KUKA KRL program: MyProgram_117().src

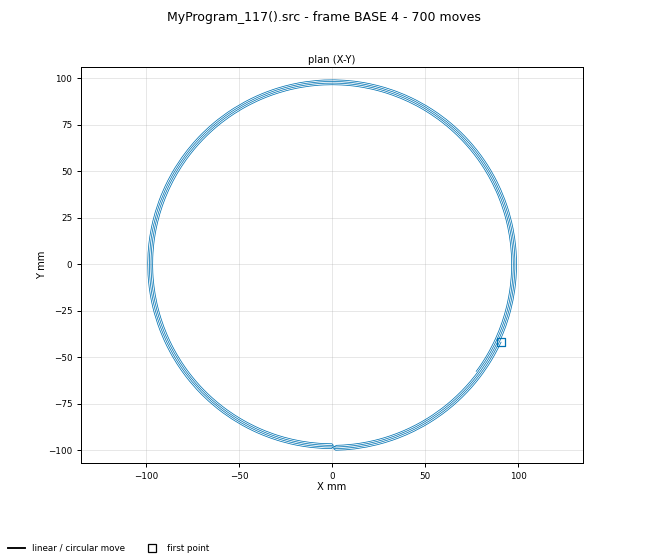
[picture p0: tool path of MyProgram_117().src in frame BASE 4, 700 of 700 moves have a stored position in this frame; points joined in program order, loops and branches not executed]
&ACCESS RVP
&REL 1
&PARAM TEMPLATE = C:\KRC\Roboter\Template\vorgabe
&PARAM EDITMASK = *
DEF MyProgram_117()
; ---- Setting reference (Base) ----
$BASE = BASE_DATA[4]

; --------------------------
; ---- Setting tool (TCP) ----
$TOOL = TOOL_DATA[3]
; --------------------------

$VEL.CP = VEL_APROX_PRINT
Startdeposition()
$VEL.CP = VEL_PRINT
LIN {X 90.8546,Y -41.8961,Z 100,A -29.5079,B 24.9354,C -1.8557,E1 25.1448,E2 114.9492} C_DIS
LIN {X 89.261,Y -45.1921,Z 100,A -32.3169,B 24.9378,C -1.821,E1 25.1412,E2 117.825} C_DIS
LIN {X 87.3886,Y -48.713,Z 100,A -34.4656,B 24.9379,C -1.8197,E1 25.1383,E2 119.9656} C_DIS
LIN {X 85.5953,Y -51.7996,Z 100,A -35.9593,B 24.9368,C -1.8357,E1 25.1362,E2 121.4139} C_DIS
LIN {X 83.9809,Y -54.379,Z 100,A -37.6896,B 24.9371,C -1.8312,E1 25.1336,E2 123.1461} C_DIS
LIN {X 81.1515,Y -58.5183,Z 100,A -40.5595,B 24.9377,C -1.8233,E1 25.129,E2 126.0206} C_DIS
LIN {X 79.2624,Y -61.0507,Z 100,A -42.3506,B 24.938,C -1.8191,E1 25.126,E2 127.813} C_DIS
LIN {X 77.0516,Y -63.8185,Z 100,A -44.3798,B 24.9383,C -1.8138,E1 25.1224,E2 129.8455} C_DIS
LIN {X 74.8748,Y -66.3606,Z 100,A -46.3784,B 24.9389,C -1.8055,E1 25.1187,E2 131.8545} C_DIS
LIN {X 72.5253,Y -68.9207,Z 100,A -48.3686,B 24.9392,C -1.8005,E1 25.1149,E2 133.8478} C_DIS
LIN {X 70.0798,Y -71.4048,Z 100,A -50.3649,B 24.9396,C -1.7957,E1 25.111,E2 135.8471} C_DIS
LIN {X 67.5259,Y -73.824,Z 100,A -52.2794,B 24.9396,C -1.7949,E1 25.1071,E2 137.7558} C_DIS
LIN {X 64.7927,Y -76.2341,Z 100,A -54.4126,B 24.9401,C -1.7883,E1 25.1026,E2 139.8962} C_DIS
LIN {X 61.8717,Y -78.6235,Z 100,A -56.541,B 24.9403,C -1.7848,E1 25.0979,E2 142.0247} C_DIS
LIN {X 59.1319,Y -80.704,Z 100,A -59.2836,B 24.9426,C -1.7507,E1 25.0916,E2 144.8383} C_DIS
LIN {X 55.2065,Y -83.4385,Z 100,A -61.177,B 24.9407,C -1.778,E1 25.0874,E2 146.6607} C_DIS
LIN {X 52.4744,Y -85.1851,Z 100,A -63.1603,B 24.9413,C -1.7695,E1 25.0827,E2 148.6577} C_DIS
LIN {X 49.4197,Y -86.9922,Z 100,A -65.3121,B 24.9419,C -1.7612,E1 25.0774,E2 150.8227} C_DIS
LIN {X 43.9764,Y -89.8668,Z 100,A -68.5455,B 24.9415,C -1.7666,E1 25.0695,E2 154.0344} C_DIS
LIN {X 39.8661,Y -91.7629,Z 100,A -71.8907,B 24.9437,C -1.7338,E1 25.0607,E2 157.4489} C_DIS
LIN {X 35.7477,Y -93.4448,Z 100,A -73.7112,B 24.9421,C -1.758,E1 25.0562,E2 159.2081} C_DIS
LIN {X 32.4545,Y -94.6398,Z 100,A -75.7667,B 24.9424,C -1.7535,E1 25.0507,E2 161.2702} C_DIS
LIN {X 28.1104,Y -96.0182,Z 100,A -78.5161,B 24.9429,C -1.7452,E1 25.0434,E2 164.0343} C_DIS
LIN {X 24.2258,Y -97.0727,Z 100,A -81.6804,B 24.9452,C -1.7105,E1 25.0346,E2 167.276} C_DIS
LIN {X 18.6579,Y -98.2938,Z 100,A -83.3794,B 24.9415,C -1.7666,E1 25.0303,E2 168.84} C_DIS
LIN {X 12.1471,Y -99.3097,Z 100,A -87.4897,B 24.9425,C -1.7511,E1 25.0189,E2 172.9832} C_DIS
LIN {X 7.1479,Y -99.7937,Z 100,A -90.5333,B 24.943,C -1.7433,E1 25.0104,E2 176.0435} C_DIS
LIN {X 1.9327,Y -100.0299,Z 100,A -93.4838,B 24.943,C -1.7437,E1 25.0021,E2 178.9923} C_DIS
LIN {X 1.9327,Y -100.0299,Z 100,A -93.4838,B 24.943,C -1.7437,E1 25.0021,E2 178.9923} C_DIS
Enddeposition()
LIN {X 0.6913,Y -99.1652,Z 100,A -93.9796,B 24.9415,C -1.767,E1 25.0009,E2 179.4329} C_DIS
Startdeposition()
$VEL.CP = VEL_PRINT
LIN {X 6.2659,Y -98.9734,Z 100,A -90.3547,B 24.9404,C -1.7829,E1 25.0111,E2 175.771} C_DIS
LIN {X 9.1996,Y -98.743,Z 100,A -88.1393,B 24.939,C -1.8033,E1 25.0174,E2 173.5087} C_DIS
LIN {X 12.9587,Y -98.3206,Z 100,A -85.2245,B 24.937,C -1.8326,E1 25.0257,E2 170.5267} C_DIS
LIN {X 18.458,Y -97.4382,Z 100,A -83.3272,B 24.9403,C -1.7846,E1 25.0306,E2 168.7453} C_DIS
LIN {X 23.319,Y -96.3902,Z 100,A -80.2469,B 24.9396,C -1.7951,E1 25.039,E2 165.6443} C_DIS
LIN {X 26.3077,Y -95.6187,Z 100,A -78.5649,B 24.9397,C -1.7931,E1 25.0435,E2 163.9697} C_DIS
LIN {X 30.9499,Y -94.2184,Z 100,A -75.585,B 24.9391,C -1.8032,E1 25.0515,E2 160.9713} C_DIS
LIN {X 34.1098,Y -93.1201,Z 100,A -73.9959,B 24.9398,C -1.7925,E1 25.0556,E2 159.4108} C_DIS
LIN {X 40.541,Y -90.5057,Z 100,A -69.6647,B 24.9386,C -1.8105,E1 25.0669,E2 155.0468} C_DIS
LIN {X 43.8774,Y -88.9361,Z 100,A -67.6389,B 24.9386,C -1.8099,E1 25.072,E2 153.0279} C_DIS
LIN {X 46.0291,Y -87.8418,Z 100,A -66.2942,B 24.9386,C -1.8103,E1 25.0753,E2 151.686} C_DIS
LIN {X 49.9401,Y -85.6805,Z 100,A -63.5045,B 24.9377,C -1.823,E1 25.0821,E2 148.8744} C_DIS
LIN {X 52.9459,Y -83.8557,Z 100,A -61.6939,B 24.938,C -1.8182,E1 25.0864,E2 147.0809} C_DIS
LIN {X 57.7115,Y -80.6487,Z 100,A -58.2792,B 24.9373,C -1.8286,E1 25.0943,E2 143.6532} C_DIS
LIN {X 59.9569,Y -78.9951,Z 100,A -56.5708,B 24.9368,C -1.8358,E1 25.0981,E2 141.9339} C_DIS
LIN {X 62.7275,Y -76.8128,Z 100,A -54.5611,B 24.9366,C -1.8392,E1 25.1025,E2 139.9238} C_DIS
LIN {X 65.4078,Y -74.5432,Z 100,A -52.5255,B 24.9363,C -1.8441,E1 25.1068,E2 137.8846} C_DIS
LIN {X 68.1055,Y -72.0868,Z 100,A -50.4771,B 24.9361,C -1.8467,E1 25.111,E2 135.8384} C_DIS
LIN {X 70.6086,Y -69.6365,Z 100,A -48.5177,B 24.9359,C -1.8491,E1 25.1149,E2 133.8817} C_DIS
LIN {X 73.1184,Y -66.9964,Z 100,A -46.4051,B 24.9355,C -1.8547,E1 25.1189,E2 131.7651} C_DIS
LIN {X 75.5655,Y -64.2237,Z 100,A -44.3231,B 24.9353,C -1.858,E1 25.1227,E2 129.6846} C_DIS
LIN {X 77.8109,Y -61.4839,Z 100,A -42.25,B 24.9348,C -1.8645,E1 25.1264,E2 127.6058} C_DIS
LIN {X 79.842,Y -58.8231,Z 100,A -40.4207,B 24.9348,C -1.8656,E1 25.1294,E2 125.7828} C_DIS
LIN {X 81.2965,Y -56.7955,Z 100,A -38.5075,B 24.9331,C -1.8885,E1 25.1326,E2 123.8247} C_DIS
LIN {X 83.0913,Y -54.1382,Z 100,A -36.9749,B 24.9337,C -1.8808,E1 25.1349,E2 122.318} C_DIS
LIN {X 84.6691,Y -51.633,Z 100,A -34.534,B 24.9312,C -1.9153,E1 25.1385,E2 119.8081} C_DIS
LIN {X 87.0569,Y -47.497,Z 100,A -32.9217,B 24.934,C -1.877,E1 25.1406,E2 118.2946} C_DIS
LIN {X 89.1564,Y -43.4308,Z 100,A -29.8964,B 24.9323,C -1.9001,E1 25.1444,E2 115.2308} C_DIS
LIN {X 90.6651,Y -40.1874,Z 100,A -27.4278,B 24.9307,C -1.9227,E1 25.1473,E2 112.7224} C_DIS
LIN {X 92.0383,Y -36.9323,Z 100,A -25.8511,B 24.9316,C -1.9101,E1 25.1489,E2 111.1841} C_DIS
LIN {X 93.3981,Y -33.3451,Z 100,A -23.5352,B 24.9308,C -1.921,E1 25.1511,E2 108.8554} C_DIS
LIN {X 95.0827,Y -28.1796,Z 100,A -20.5952,B 24.9307,C -1.9228,E1 25.1536,E2 105.9278} C_DIS
LIN {X 95.9761,Y -24.9697,Z 100,A -18.685,B 24.9303,C -1.9283,E1 25.155,E2 104.0156} C_DIS
LIN {X 97.2767,Y -19.2966,Z 100,A -15.4761,B 24.93,C -1.9328,E1 25.1569,E2 100.8147} C_DIS
LIN {X 98.201,Y -13.834,Z 100,A -12.0909,B 24.9287,C -1.9505,E1 25.1585,E2 97.4077} C_DIS
LIN {X 98.5903,Y -10.7206,Z 100,A -9.9416,B 24.9272,C -1.97,E1 25.1591,E2 95.2251} C_DIS
LIN {X 98.886,Y -7.5176,Z 100,A -7.8658,B 24.9261,C -1.9849,E1 25.1595,E2 93.1265} C_DIS
LIN {X 99.1121,Y -3.4295,Z 100,A -6.1235,B 24.9274,C -1.9672,E1 25.1597,E2 91.4364} C_DIS
LIN {X 99.1305,Y 2.8285,Z 100,A -1.9325,B 24.9248,C -2.0022,E1 25.1596,E2 87.1877} C_DIS
LIN {X 98.9312,Y 6.8905,Z 100,A -0.1687,B 24.9261,C -1.9859,E1 25.1593,E2 85.4728} C_DIS
LIN {X 98.7353,Y 9.2834,Z 100,A 1.9576,B 24.9235,C -2.0204,E1 25.1587,E2 83.2778} C_DIS
LIN {X 98.1786,Y 13.9922,Z 100,A 3.4043,B 24.9267,C -1.9767,E1 25.1582,E2 81.9425} C_DIS
LIN {X 97.3147,Y 19.0993,Z 100,A 6.8499,B 24.9247,C -2.0042,E1 25.1565,E2 78.4524} C_DIS
LIN {X 96.5792,Y 22.5236,Z 100,A 9.8653,B 24.9211,C -2.0507,E1 25.1546,E2 75.3448} C_DIS
LIN {X 95.1729,Y 27.8757,Z 100,A 12.0003,B 24.9237,C -2.0174,E1 25.153,E2 73.3006} C_DIS
LIN {X 94.2802,Y 30.7591,Z 100,A 13.8408,B 24.923,C -2.0265,E1 25.1514,E2 71.449} C_DIS
LIN {X 92.9322,Y 34.6224,Z 100,A 16.1677,B 24.9226,C -2.032,E1 25.1492,E2 69.1222} C_DIS
LIN {X 90.6792,Y 40.1549,Z 100,A 19.4045,B 24.9225,C -2.0334,E1 25.1458,E2 65.8999} C_DIS
LIN {X 88.6792,Y 44.3956,Z 100,A 22.1934,B 24.9216,C -2.0442,E1 25.1424,E2 63.1005} C_DIS
LIN {X 87.2725,Y 47.0996,Z 100,A 24.1381,B 24.9207,C -2.0563,E1 25.1398,E2 61.1374} C_DIS
LIN {X 85.3146,Y 50.5593,Z 100,A 26.3186,B 24.9206,C -2.0579,E1 25.1368,E2 58.9645} C_DIS
LIN {X 83.6341,Y 53.2941,Z 100,A 28.1593,B 24.9203,C -2.0622,E1 25.134,E2 57.1229} C_DIS
LIN {X 82.0137,Y 55.7549,Z 100,A 30.2378,B 24.9188,C -2.0814,E1 25.1307,E2 55.0092} C_DIS
LIN {X 80.1035,Y 58.466,Z 100,A 31.6874,B 24.9198,C -2.0677,E1 25.1284,E2 53.599} C_DIS
LIN {X 77.9344,Y 61.3277,Z 100,A 33.816,B 24.9193,C -2.0749,E1 25.1248,E2 51.4636} C_DIS
LIN {X 75.5962,Y 64.1876,Z 100,A 35.6617,B 24.9198,C -2.0686,E1 25.1215,E2 49.6412} C_DIS
LIN {X 73.8444,Y 66.1954,Z 100,A 37.9636,B 24.9171,C -2.102,E1 25.1171,E2 47.2706} C_DIS
LIN {X 71.3218,Y 68.906,Z 100,A 39.5535,B 24.9185,C -2.0851,E1 25.1141,E2 45.7275} C_DIS
LIN {X 69.2349,Y 71.0047,Z 100,A 41.4391,B 24.9176,C -2.0956,E1 25.1103,E2 43.8251} C_DIS
LIN {X 66.2722,Y 73.7756,Z 100,A 43.5685,B 24.9179,C -2.092,E1 25.106,E2 41.7128} C_DIS
LIN {X 63.6338,Y 76.0636,Z 100,A 45.9997,B 24.9163,C -2.112,E1 25.1007,E2 39.2438} C_DIS
LIN {X 61.144,Y 78.0795,Z 100,A 48.2904,B 24.9147,C -2.1325,E1 25.0956,E2 36.913} C_DIS
LIN {X 57.2387,Y 80.9861,Z 100,A 50.1264,B 24.9173,C -2.0994,E1 25.0916,E2 35.1617} C_DIS
LIN {X 54.0365,Y 83.1576,Z 100,A 52.6018,B 24.9163,C -2.1123,E1 25.0858,E2 32.6641} C_DIS
LIN {X 50.8122,Y 85.1651,Z 100,A 54.7198,B 24.9163,C -2.1126,E1 25.0808,E2 30.5519} C_DIS
LIN {X 45.3585,Y 88.19,Z 100,A 58.2162,B 24.9163,C -2.1134,E1 25.0722,E2 27.0637} C_DIS
LIN {X 42.553,Y 89.5782,Z 100,A 60.1676,B 24.9156,C -2.1211,E1 25.0673,E2 25.0993} C_DIS
LIN {X 38.7954,Y 91.2679,Z 100,A 62.5974,B 24.9153,C -2.1256,E1 25.061,E2 22.6647} C_DIS
LIN {X 35.0727,Y 92.7616,Z 100,A 64.7142,B 24.9157,C -2.1203,E1 25.0556,E2 20.5651} C_DIS
LIN {X 32.749,Y 93.6073,Z 100,A 66.4711,B 24.9146,C -2.1339,E1 25.0509,E2 18.7794} C_DIS
LIN {X 28.3562,Y 95.0303,Z 100,A 68.8789,B 24.9152,C -2.1262,E1 25.0445,E2 16.3944} C_DIS
LIN {X 24.5316,Y 96.0887,Z 100,A 71.9667,B 24.9127,C -2.1575,E1 25.036,E2 13.2371} C_DIS
LIN {X 19.8131,Y 97.1714,Z 100,A 73.8566,B 24.9153,C -2.1249,E1 25.031,E2 11.427} C_DIS
LIN {X 16.7703,Y 97.7433,Z 100,A 75.4869,B 24.9157,C -2.1197,E1 25.0266,E2 9.8108} C_DIS
LIN {X 12.2429,Y 98.4133,Z 100,A 78.5022,B 24.9146,C -2.134,E1 25.0182,E2 6.7641} C_DIS
LIN {X 7.0795,Y 98.9184,Z 100,A 81.1159,B 24.9157,C -2.1202,E1 25.011,E2 4.1847} C_DIS
LIN {X 1.4329,Y 99.1611,Z 100,A 84.378,B 24.9157,C -2.1198,E1 25.0019,E2 0.9244} C_DIS
LIN {X -4.0931,Y 99.0863,Z 100,A 87.4521,B 24.9161,C -2.1146,E1 24.9934,E2 -2.1376} C_DIS
LIN {X -7.6767,Y 98.8733,Z 100,A 90.1777,B 24.9143,C -2.1373,E1 24.9856,E2 -4.9181} C_DIS
LIN {X -14.3965,Y 98.1211,Z 100,A 93.8164,B 24.9153,C -2.1253,E1 24.9756,E2 -8.5308} C_DIS
LIN {X -17.8618,Y 97.5493,Z 100,A 96.4541,B 24.9137,C -2.1457,E1 24.9682,E2 -11.2196} C_DIS
LIN {X -21.8344,Y 96.7384,Z 100,A 97.9981,B 24.9161,C -2.115,E1 24.9642,E2 -12.6926} C_DIS
LIN {X -25.5325,Y 95.8281,Z 100,A 100.4259,B 24.9156,C -2.1209,E1 24.9576,E2 -15.1379} C_DIS
LIN {X -29.0848,Y 94.8102,Z 100,A 102.2357,B 24.9167,C -2.1071,E1 24.9528,E2 -16.9178} C_DIS
LIN {X -31.6314,Y 93.9908,Z 100,A 104.1295,B 24.9159,C -2.1175,E1 24.9477,E2 -18.84} C_DIS
LIN {X -35.1644,Y 92.7269,Z 100,A 106.1336,B 24.9166,C -2.1089,E1 24.9425,E2 -20.8278} C_DIS
LIN {X -37.7966,Y 91.6861,Z 100,A 107.8796,B 24.9165,C -2.1105,E1 24.9379,E2 -22.5814} C_DIS
LIN {X -40.7171,Y 90.4264,Z 100,A 110.1476,B 24.9155,C -2.123,E1 24.9321,E2 -24.8844} C_DIS
LIN {X -43.672,Y 89.0374,Z 100,A 111.6554,B 24.9168,C -2.1067,E1 24.9284,E2 -26.3574} C_DIS
LIN {X -46.915,Y 87.3726,Z 100,A 113.5154,B 24.9177,C -2.0946,E1 24.9238,E2 -28.1937} C_DIS
LIN {X -53.0828,Y 83.7697,Z 100,A 117.9867,B 24.9174,C -2.0989,E1 24.9131,E2 -32.6891} C_DIS
LIN {X -56.3961,Y 81.574,Z 100,A 120.2522,B 24.9178,C -2.0934,E1 24.9078,E2 -34.9489} C_DIS
LIN {X -61.3368,Y 77.9272,Z 100,A 123.7519,B 24.9185,C -2.0843,E1 24.9,E2 -38.4395} C_DIS
LIN {X -63.4455,Y 76.22,Z 100,A 125.9799,B 24.917,C -2.1036,E1 24.8951,E2 -40.722} C_DIS
LIN {X -66.6139,Y 73.4693,Z 100,A 128.4285,B 24.9174,C -2.0988,E1 24.8901,E2 -43.169} C_DIS
LIN {X -69.5784,Y 70.666,Z 100,A 130.0947,B 24.9197,C -2.0695,E1 24.8869,E2 -44.7722} C_DIS
LIN {X -71.8411,Y 68.3668,Z 100,A 132.6576,B 24.9182,C -2.0888,E1 24.8818,E2 -47.3923} C_DIS
LIN {X -74.5581,Y 65.3907,Z 100,A 134.5074,B 24.9199,C -2.0665,E1 24.8785,E2 -49.1973} C_DIS
LIN {X -77.9352,Y 61.3267,Z 100,A 137.3121,B 24.9212,C -2.0501,E1 24.8736,E2 -51.9759} C_DIS
LIN {X -80.8016,Y 57.4972,Z 100,A 140.3008,B 24.9212,C -2.0502,E1 24.8686,E2 -54.9793} C_DIS
LIN {X -84.438,Y 52.0134,Z 100,A 144.0835,B 24.9221,C -2.0388,E1 24.8629,E2 -58.7539} C_DIS
LIN {X -86.0785,Y 49.2477,Z 100,A 146.7197,B 24.9204,C -2.0599,E1 24.8591,E2 -61.4541} C_DIS
LIN {X -88.337,Y 45.071,Z 100,A 148.636,B 24.9232,C -2.0238,E1 24.8568,E2 -63.2946} C_DIS
LIN {X -89.8728,Y 41.925,Z 100,A 150.3939,B 24.9243,C -2.0089,E1 24.8547,E2 -65.0264} C_DIS
LIN {X -91.9957,Y 37.0345,Z 100,A 154.0806,B 24.9235,C -2.0198,E1 24.8506,E2 -68.7595} C_DIS
LIN {X -93.141,Y 34.0526,Z 100,A 156.8724,B 24.9215,C -2.0462,E1 24.8479,E2 -71.6302} C_DIS
LIN {X -95.0967,Y 28.1325,Z 100,A 158.9789,B 24.9262,C -1.9844,E1 24.8463,E2 -73.6012} C_DIS
LIN {X -96.3633,Y 23.4293,Z 100,A 162.1051,B 24.9261,C -1.9858,E1 24.844,E2 -76.7492} C_DIS
LIN {X -97.147,Y 19.9317,Z 100,A 164.1597,B 24.9266,C -1.9787,E1 24.8428,E2 -78.7988} C_DIS
LIN {X -98.0211,Y 15.0562,Z 100,A 167.0727,B 24.9271,C -1.9712,E1 24.8415,E2 -81.7113} C_DIS
LIN {X -98.5567,Y 11.0293,Z 100,A 170.3255,B 24.9254,C -1.9941,E1 24.8404,E2 -85.0382} C_DIS
LIN {X -98.9855,Y 6.0807,Z 100,A 172.357,B 24.9282,C -1.9566,E1 24.84,E2 -86.9924} C_DIS
LIN {X -99.1342,Y 2.7095,Z 100,A 174.2253,B 24.9289,C -1.9476,E1 24.8398,E2 -88.8505} C_DIS
LIN {X -99.1684,Y 0.6951,Z 100,A 175.7702,B 24.9282,C -1.9566,E1 24.8398,E2 -90.4262} C_DIS
LIN {X -99.0153,Y -5.5482,Z 100,A 179.0512,B 24.9299,C -1.9341,E1 24.8401,E2 -93.6731} C_DIS
LIN {X -98.7637,Y -8.9753,Z 100,A -178.3436,B 24.9288,C -1.9486,E1 24.8408,E2 -96.3287} C_DIS
LIN {X -98.3563,Y -12.6829,Z 100,A -176.6482,B 24.9304,C -1.9263,E1 24.8413,E2 -97.981} C_DIS
LIN {X -97.8334,Y -16.2313,Z 100,A -174.6127,B 24.931,C -1.9185,E1 24.8422,E2 -100.0101} C_DIS
LIN {X -97.2266,Y -19.544,Z 100,A -172.613,B 24.9313,C -1.9143,E1 24.8433,E2 -102.0114} C_DIS
LIN {X -96.4078,Y -23.2471,Z 100,A -170.4736,B 24.9319,C -1.9058,E1 24.8446,E2 -104.1431} C_DIS
LIN {X -95.661,Y -26.151,Z 100,A -168.6012,B 24.9319,C -1.9052,E1 24.846,E2 -106.0251} C_DIS
LIN {X -93.8161,Y -32.1464,Z 100,A -165.0105,B 24.9328,C -1.8932,E1 24.849,E2 -109.6076} C_DIS
LIN {X -92.5501,Y -35.6314,Z 100,A -161.8525,B 24.9308,C -1.9216,E1 24.8523,E2 -112.8513} C_DIS
LIN {X -90.3767,Y -40.8274,Z 100,A -159.6526,B 24.934,C -1.8762,E1 24.8546,E2 -114.955} C_DIS
LIN {X -88.9026,Y -43.9448,Z 100,A -157.6433,B 24.9344,C -1.8712,E1 24.8571,E2 -116.9632} C_DIS
LIN {X -87.2503,Y -47.1404,Z 100,A -155.5837,B 24.9348,C -1.8648,E1 24.8598,E2 -119.0186} C_DIS
LIN {X -85.9838,Y -49.4125,Z 100,A -153.8216,B 24.9345,C -1.8697,E1 24.8622,E2 -120.8013} C_DIS
LIN {X -83.428,Y -53.6152,Z 100,A -150.9996,B 24.935,C -1.8616,E1 24.8664,E2 -123.6184} C_DIS
LIN {X -81.1676,Y -56.9811,Z 100,A -148.8483,B 24.9359,C -1.8491,E1 24.8698,E2 -125.7505} C_DIS
LIN {X -78.917,Y -60.0583,Z 100,A -146.3568,B 24.9356,C -1.8536,E1 24.874,E2 -128.2649} C_DIS
LIN {X -76.6092,Y -62.9772,Z 100,A -143.3514,B 24.9338,C -1.8785,E1 24.8795,E2 -131.3435} C_DIS
LIN {X -72.8133,Y -67.3289,Z 100,A -141.0169,B 24.9368,C -1.8359,E1 24.8837,E2 -133.5869} C_DIS
LIN {X -70.4028,Y -69.8449,Z 100,A -138.0223,B 24.9347,C -1.8662,E1 24.8898,E2 -136.6663} C_DIS
LIN {X -66.3283,Y -73.7253,Z 100,A -135.8013,B 24.9377,C -1.8232,E1 24.8941,E2 -138.7941} C_DIS
LIN {X -61.8773,Y -77.5,Z 100,A -132.2172,B 24.9377,C -1.8243,E1 24.9019,E2 -142.3943} C_DIS
LIN {X -58.6752,Y -79.9503,Z 100,A -129.7231,B 24.9375,C -1.8261,E1 24.9075,E2 -144.9016} C_DIS
LIN {X -53.7609,Y -83.3345,Z 100,A -126.6443,B 24.9388,C -1.8075,E1 24.9145,E2 -147.9462} C_DIS
LIN {X -48.5279,Y -86.4864,Z 100,A -123.0861,B 24.939,C -1.8034,E1 24.9231,E2 -151.5055} C_DIS
LIN {X -45.4862,Y -88.1248,Z 100,A -121.0314,B 24.939,C -1.8029,E1 24.9282,E2 -153.5647} C_DIS
LIN {X -42.6776,Y -89.5183,Z 100,A -119.3698,B 24.9396,C -1.7953,E1 24.9323,E2 -155.2127} C_DIS
LIN {X -40.5018,Y -90.5234,Z 100,A -117.7985,B 24.9392,C -1.8005,E1 24.9363,E2 -156.8001} C_DIS
LIN {X -37.1909,Y -91.9331,Z 100,A -115.8808,B 24.9398,C -1.7925,E1 24.9413,E2 -158.7032} C_DIS
LIN {X -33.2428,Y -93.4333,Z 100,A -113.2446,B 24.9394,C -1.7974,E1 24.9482,E2 -161.3564} C_DIS
LIN {X -29.3727,Y -94.7209,Z 100,A -111.0463,B 24.94,C -1.7899,E1 24.954,E2 -163.5408} C_DIS
LIN {X -27.2455,Y -95.3548,Z 100,A -108.7966,B 24.9376,C -1.8246,E1 24.9603,E2 -165.8764} C_DIS
LIN {X -22.3273,Y -96.6245,Z 100,A -106.7888,B 24.94,C -1.7888,E1 24.9655,E2 -167.8019} C_DIS
LIN {X -19.3944,Y -97.2573,Z 100,A -104.4465,B 24.9386,C -1.8105,E1 24.9721,E2 -170.1985} C_DIS
LIN {X -15.6093,Y -97.9356,Z 100,A -102.0586,B 24.9382,C -1.8161,E1 24.9787,E2 -172.6019} C_DIS
LIN {X -11.1761,Y -98.5395,Z 100,A -100.1508,B 24.9399,C -1.7905,E1 24.9838,E2 -174.4501} C_DIS
LIN {X -4.9792,Y -99.0465,Z 100,A -96.6781,B 24.9402,C -1.786,E1 24.9935,E2 -177.9135} C_DIS
LIN {X -0.5004,Y -99.1694,Z 100,A -94.031,B 24.94,C -1.7886,E1 25.0009,E2 -180.5671} C_DIS
LIN {X -0.5004,Y -99.1694,Z 100,A -94.031,B 24.94,C -1.7886,E1 25.0009,E2 -180.5671} C_DIS
Enddeposition()
LIN {X 0.7031,Y -98.2806,Z 100,A -94.8995,B 24.9428,C -1.7469,E1 24.9982,E2 -179.5997} C_DIS
Startdeposition()
$VEL.CP = VEL_PRINT
LIN {X -3.7844,Y -98.2208,Z 100,A -96.6689,B 24.9408,C -1.777,E1 24.9935,E2 -177.9015} C_DIS
LIN {X -9.0806,Y -97.8724,Z 100,A -99.5035,B 24.9402,C -1.7864,E1 24.9856,E2 -175.088} C_DIS
LIN {X -12.0024,Y -97.5572,Z 100,A -101.792,B 24.9416,C -1.7658,E1 24.9791,E2 -172.7492} C_DIS
LIN {X -15.3506,Y -97.0872,Z 100,A -103.9453,B 24.942,C -1.7597,E1 24.9731,E2 -170.5797} C_DIS
LIN {X -19.3218,Y -96.376,Z 100,A -105.9871,B 24.9412,C -1.7717,E1 24.9676,E2 -168.5641} C_DIS
LIN {X -22.607,Y -95.6589,Z 100,A -108.4713,B 24.9423,C -1.7541,E1 24.9607,E2 -166.0347} C_DIS
LIN {X -25.966,Y -94.8016,Z 100,A -109.8291,B 24.9407,C -1.7788,E1 24.9572,E2 -164.7335} C_DIS
LIN {X -28.3424,Y -94.1187,Z 100,A -111.4726,B 24.9411,C -1.7726,E1 24.9528,E2 -163.0726} C_DIS
LIN {X -31.6213,Y -93.0677,Z 100,A -114.2445,B 24.9428,C -1.7474,E1 24.9453,E2 -160.2357} C_DIS
LIN {X -35.9301,Y -91.4903,Z 100,A -116.1039,B 24.9407,C -1.7784,E1 24.9406,E2 -158.4459} C_DIS
LIN {X -40.2807,Y -89.6601,Z 100,A -118.9222,B 24.9407,C -1.779,E1 24.9334,E2 -155.6224} C_DIS
LIN {X -43.3286,Y -88.2282,Z 100,A -120.8746,B 24.9405,C -1.7816,E1 24.9284,E2 -153.6714} C_DIS
LIN {X -46.1911,Y -86.7642,Z 100,A -122.6869,B 24.9402,C -1.7862,E1 24.924,E2 -151.8649} C_DIS
LIN {X -48.8551,Y -85.2916,Z 100,A -124.7909,B 24.9408,C -1.7773,E1 24.9188,E2 -149.7336} C_DIS
LIN {X -52.593,Y -83.0409,Z 100,A -127.2914,B 24.9404,C -1.7825,E1 24.9129,E2 -147.2378} C_DIS
LIN {X -56.3842,Y -80.5133,Z 100,A -129.9455,B 24.9401,C -1.787,E1 24.9068,E2 -144.5853} C_DIS
LIN {X -59.6748,Y -78.106,Z 100,A -133.5265,B 24.9426,C -1.7506,E1 24.8986,E2 -140.9047} C_DIS
LIN {X -64.9815,Y -73.7499,Z 100,A -135.4992,B 24.9374,C -1.8268,E1 24.8948,E2 -139.1058} C_DIS
LIN {X -70.1765,Y -68.8247,Z 100,A -140.036,B 24.9377,C -1.8228,E1 24.8855,E2 -134.5407} C_DIS
LIN {X -75.4021,Y -63.0561,Z 100,A -144.6109,B 24.9371,C -1.8317,E1 24.877,E2 -129.9666} C_DIS
LIN {X -79.3284,Y -58.0385,Z 100,A -148.5605,B 24.9371,C -1.8327,E1 24.8702,E2 -126.0007} C_DIS
LIN {X -81.2404,Y -55.331,Z 100,A -150.6432,B 24.9371,C -1.8325,E1 24.8668,E2 -123.9073} C_DIS
LIN {X -82.7159,Y -53.0993,Z 100,A -152.646,B 24.9378,C -1.8219,E1 24.8638,E2 -121.8691} C_DIS
LIN {X -84.5723,Y -50.0898,Z 100,A -154.1854,B 24.9362,C -1.8446,E1 24.8616,E2 -120.3758} C_DIS
LIN {X -85.8025,Y -47.952,Z 100,A -155.6566,B 24.936,C -1.8473,E1 24.8596,E2 -118.9035} C_DIS
LIN {X -87.4778,Y -44.8231,Z 100,A -157.7262,B 24.9356,C -1.853,E1 24.8569,E2 -116.8363} C_DIS
LIN {X -89.0012,Y -41.717,Z 100,A -159.7411,B 24.9352,C -1.8587,E1 24.8545,E2 -114.8241} C_DIS
LIN {X -91.1623,Y -36.7559,Z 100,A -162.6115,B 24.9339,C -1.8771,E1 24.8514,E2 -111.9818} C_DIS
LIN {X -92.5847,Y -33.0118,Z 100,A -165.735,B 24.9353,C -1.8581,E1 24.8483,E2 -108.7953} C_DIS
LIN {X -93.6148,Y -29.9623,Z 100,A -167.1224,B 24.9338,C -1.8796,E1 24.8471,E2 -107.4514} C_DIS
LIN {X -94.3373,Y -27.6054,Z 100,A -168.7403,B 24.9338,C -1.8781,E1 24.8458,E2 -105.8204} C_DIS
LIN {X -95.2127,Y -24.4133,Z 100,A -170.5413,B 24.9332,C -1.8882,E1 24.8445,E2 -104.033} C_DIS
LIN {X -96.017,Y -21.0287,Z 100,A -172.6216,B 24.9328,C -1.8927,E1 24.8432,E2 -101.9513} C_DIS
LIN {X -96.7295,Y -17.4606,Z 100,A -174.7143,B 24.9323,C -1.9002,E1 24.8421,E2 -99.8642} C_DIS
LIN {X -97.214,Y -14.5307,Z 100,A -176.6315,B 24.9323,C -1.8996,E1 24.8413,E2 -97.9341} C_DIS
LIN {X -97.7927,Y -9.9071,Z 100,A -179.13,B 24.9312,C -1.9153,E1 24.8405,E2 -95.4581} C_DIS
LIN {X -98.0751,Y -6.5381,Z 100,A 178.7822,B 24.931,C -1.9178,E1 24.8401,E2 -93.3636} C_DIS
LIN {X -98.2689,Y -2.1956,Z 100,A 176.167,B 24.9307,C -1.9233,E1 24.8398,E2 -90.7458} C_DIS
LIN {X -98.2774,Y 1.7359,Z 100,A 173.9513,B 24.9299,C -1.9331,E1 24.8398,E2 -88.5403} C_DIS
LIN {X -98.1668,Y 4.9918,Z 100,A 171.8896,B 24.9299,C -1.9339,E1 24.8401,E2 -86.468} C_DIS
LIN {X -97.7338,Y 10.4695,Z 100,A 168.7137,B 24.9291,C -1.9451,E1 24.8409,E2 -83.2999} C_DIS
LIN {X -97.2936,Y 13.9796,Z 100,A 166.2454,B 24.9295,C -1.9387,E1 24.8418,E2 -80.8014} C_DIS
LIN {X -96.7553,Y 17.3167,Z 100,A 164.5822,B 24.9284,C -1.9549,E1 24.8426,E2 -79.167} C_DIS
LIN {X -96.0221,Y 21.0051,Z 100,A 162.5374,B 24.9275,C -1.9666,E1 24.8438,E2 -77.1382} C_DIS
LIN {X -94.3008,Y 27.7287,Z 100,A 157.9594,B 24.9278,C -1.9622,E1 24.8471,E2 -72.523} C_DIS
LIN {X -93.2688,Y 31.023,Z 100,A 156.3612,B 24.9264,C -1.9819,E1 24.8485,E2 -70.9626} C_DIS
LIN {X -92.3152,Y 33.7546,Z 100,A 154.6854,B 24.9259,C -1.9874,E1 24.8501,E2 -69.2905} C_DIS
LIN {X -89.5641,Y 40.4937,Z 100,A 150.7004,B 24.9243,C -2.0087,E1 24.8543,E2 -65.3343} C_DIS
LIN {X -88.5287,Y 42.7101,Z 100,A 149.0427,B 24.9246,C -2.0054,E1 24.8563,E2 -63.6597} C_DIS
LIN {X -86.1069,Y 47.4057,Z 100,A 146.0899,B 24.9236,C -2.0186,E1 24.8601,E2 -60.7225} C_DIS
LIN {X -84.5142,Y 50.1881,Z 100,A 143.9706,B 24.9238,C -2.0158,E1 24.8631,E2 -58.5855} C_DIS
LIN {X -81.842,Y 54.438,Z 100,A 140.8042,B 24.9238,C -2.0162,E1 24.8679,E2 -55.4042} C_DIS
LIN {X -78.4434,Y 59.2297,Z 100,A 137.8768,B 24.9218,C -2.0418,E1 24.8726,E2 -52.5236} C_DIS
LIN {X -76.4122,Y 61.8275,Z 100,A 135.6842,B 24.9221,C -2.038,E1 24.8765,E2 -50.3115} C_DIS
LIN {X -74.175,Y 64.4948,Z 100,A 132.7502,B 24.924,C -2.0136,E1 24.882,E2 -47.3061} C_DIS
LIN {X -70.7666,Y 68.2169,Z 100,A 130.8743,B 24.9207,C -2.0559,E1 24.8854,E2 -45.5228} C_DIS
LIN {X -67.8558,Y 71.1124,Z 100,A 128.1822,B 24.9211,C -2.0517,E1 24.8908,E2 -42.8094} C_DIS
LIN {X -64.4484,Y 74.2155,Z 100,A 125.3056,B 24.9211,C -2.0515,E1 24.8968,E2 -39.921} C_DIS
LIN {X -60.7855,Y 77.2437,Z 100,A 122.4919,B 24.9207,C -2.0561,E1 24.9029,E2 -37.1076} C_DIS
LIN {X -57.327,Y 79.8446,Z 100,A 120.5242,B 24.9189,C -2.0798,E1 24.9073,E2 -35.1896} C_DIS
LIN {X -55.6186,Y 81.0455,Z 100,A 119.052,B 24.9194,C -2.0737,E1 24.9107,E2 -33.6977} C_DIS
LIN {X -52.9883,Y 82.7871,Z 100,A 117.2874,B 24.9189,C -2.0797,E1 24.9148,E2 -31.9417} C_DIS
LIN {X -47.8568,Y 85.8556,Z 100,A 113.838,B 24.9183,C -2.0872,E1 24.9231,E2 -28.4997} C_DIS
LIN {X -45.2856,Y 87.2411,Z 100,A 111.7097,B 24.9192,C -2.0756,E1 24.9284,E2 -26.3379} C_DIS
LIN {X -40.5076,Y 89.5578,Z 100,A 109.2375,B 24.9172,C -2.1017,E1 24.9345,E2 -23.9214} C_DIS
LIN {X -37.5307,Y 90.8469,Z 100,A 106.9552,B 24.918,C -2.091,E1 24.9405,E2 -21.6084} C_DIS
LIN {X -34.28,Y 92.123,Z 100,A 104.6053,B 24.9186,C -2.0829,E1 24.9466,E2 -19.2344} C_DIS
LIN {X -30.2573,Y 93.5198,Z 100,A 102.7517,B 24.9167,C -2.1075,E1 24.9514,E2 -17.4359} C_DIS
LIN {X -27.899,Y 94.2502,Z 100,A 101.0737,B 24.9172,C -2.1009,E1 24.9559,E2 -15.7392} C_DIS
LIN {X -24.9823,Y 95.0664,Z 100,A 99.0955,B 24.9177,C -2.0953,E1 24.9613,E2 -13.7448} C_DIS
LIN {X -22.0446,Y 95.7888,Z 100,A 97.2058,B 24.9179,C -2.0926,E1 24.9665,E2 -11.8461} C_DIS
LIN {X -17.9671,Y 96.6384,Z 100,A 94.9122,B 24.9174,C -2.0992,E1 24.9727,E2 -9.5656} C_DIS
LIN {X -14.1589,Y 97.2682,Z 100,A 92.4639,B 24.9178,C -2.0939,E1 24.9795,E2 -7.1025} C_DIS
LIN {X -7.0121,Y 98.043,Z 100,A 88.6789,B 24.9165,C -2.1102,E1 24.99,E2 -3.3542} C_DIS
LIN {X -4.124,Y 98.2062,Z 100,A 86.2458,B 24.9185,C -2.0845,E1 24.9969,E2 -0.8597} C_DIS
LIN {X 0.1184,Y 98.2938,Z 100,A 84.6375,B 24.9161,C -2.1155,E1 25.0012,E2 0.675} C_DIS
LIN {X 5.3634,Y 98.1463,Z 100,A 81.6636,B 24.9158,C -2.1188,E1 25.0095,E2 3.6404} C_DIS
LIN {X 10.6573,Y 97.7142,Z 100,A 78.3393,B 24.9165,C -2.1103,E1 25.0188,E2 6.983} C_DIS
LIN {X 14.5406,Y 97.2121,Z 100,A 75.9614,B 24.9168,C -2.1064,E1 25.0254,E2 9.3684} C_DIS
LIN {X 18.1007,Y 96.613,Z 100,A 73.7692,B 24.9171,C -2.1024,E1 25.0314,E2 11.5675} C_DIS
LIN {X 23.3318,Y 95.4834,Z 100,A 70.8393,B 24.9167,C -2.1077,E1 25.0393,E2 14.481} C_DIS
LIN {X 26.7547,Y 94.5814,Z 100,A 68.7627,B 24.9168,C -2.1058,E1 25.0449,E2 16.5586} C_DIS
LIN {X 32.5393,Y 92.7505,Z 100,A 65.293,B 24.9168,C -2.1054,E1 25.0542,E2 20.0227} C_DIS
LIN {X 35.4757,Y 91.6686,Z 100,A 63.249,B 24.9176,C -2.0956,E1 25.0595,E2 22.0856} C_DIS
LIN {X 38.5242,Y 90.4295,Z 100,A 61.5725,B 24.9171,C -2.1025,E1 25.0638,E2 23.7419} C_DIS
LIN {X 41.7358,Y 88.9925,Z 100,A 59.5129,B 24.9173,C -2.0998,E1 25.069,E2 25.8027} C_DIS
LIN {X 44.4942,Y 87.6458,Z 100,A 57.715,B 24.9175,C -2.0972,E1 25.0735,E2 27.6019} C_DIS
LIN {X 48.3497,Y 85.5804,Z 100,A 55.2562,B 24.9175,C -2.0972,E1 25.0796,E2 30.0539} C_DIS
LIN {X 50.5089,Y 84.3246,Z 100,A 53.2525,B 24.9193,C -2.0746,E1 25.0845,E2 32.1046} C_DIS
LIN {X 55.3469,Y 81.2296,Z 100,A 50.2955,B 24.9186,C -2.0838,E1 25.0913,E2 35.03} C_DIS
LIN {X 61.5543,Y 76.6319,Z 100,A 45.6992,B 24.9195,C -2.0723,E1 25.1016,E2 39.6369} C_DIS
LIN {X 65.1812,Y 73.5739,Z 100,A 43.0592,B 24.9195,C -2.0716,E1 25.1071,E2 42.2682} C_DIS
LIN {X 67.4662,Y 71.4829,Z 100,A 41.3382,B 24.9195,C -2.0712,E1 25.1106,E2 43.9834} C_DIS
LIN {X 69.1978,Y 69.808,Z 100,A 39.8013,B 24.9202,C -2.0632,E1 25.1137,E2 45.5327} C_DIS
LIN {X 73.7304,Y 65.0039,Z 100,A 36.2402,B 24.92,C -2.0656,E1 25.1205,E2 49.0723} C_DIS
LIN {X 75.1292,Y 63.382,Z 100,A 34.6532,B 24.9212,C -2.0498,E1 25.1234,E2 50.6896} C_DIS
LIN {X 77.4684,Y 60.5015,Z 100,A 32.5906,B 24.9213,C -2.0484,E1 25.127,E2 52.7457} C_DIS
LIN {X 79.4717,Y 57.8427,Z 100,A 30.1291,B 24.9232,C -2.0237,E1 25.1311,E2 55.2537} C_DIS
LIN {X 81.7242,Y 54.6165,Z 100,A 27.9606,B 24.9232,C -2.0226,E1 25.1345,E2 57.4142} C_DIS
LIN {X 83.551,Y 51.7766,Z 100,A 26.6735,B 24.9217,C -2.0437,E1 25.1363,E2 58.645} C_DIS
LIN {X 84.9275,Y 49.4888,Z 100,A 24.768,B 24.923,C -2.026,E1 25.139,E2 60.5824} C_DIS
LIN {X 86.6968,Y 46.3184,Z 100,A 22.8747,B 24.9228,C -2.0289,E1 25.1415,E2 62.459} C_DIS
LIN {X 88.02,Y 43.7486,Z 100,A 20.8751,B 24.9241,C -2.012,E1 25.1441,E2 64.4878} C_DIS
LIN {X 90.8782,Y 37.4539,Z 100,A 17.1179,B 24.9241,C -2.011,E1 25.1483,E2 68.2267} C_DIS
LIN {X 92.1336,Y 34.2506,Z 100,A 15.0035,B 24.9249,C -2.0009,E1 25.1504,E2 70.3533} C_DIS
LIN {X 93.5372,Y 30.2034,Z 100,A 12.7575,B 24.9248,C -2.0033,E1 25.1524,E2 72.5811} C_DIS
LIN {X 94.419,Y 27.3279,Z 100,A 10.3232,B 24.9271,C -1.9714,E1 25.1544,E2 75.0767} C_DIS
LIN {X 95.4247,Y 23.5724,Z 100,A 8.6089,B 24.9261,C -1.9859,E1 25.1555,E2 76.7467} C_DIS
LIN {X 96.1788,Y 20.2823,Z 100,A 6.6164,B 24.9266,C -1.9788,E1 25.1567,E2 78.7444} C_DIS
LIN {X 97.1257,Y 15.102,Z 100,A 3.7878,B 24.9266,C -1.9787,E1 25.158,E2 81.5568} C_DIS
LIN {X 97.8014,Y 9.8148,Z 100,A 0.7369,B 24.9272,C -1.971,E1 25.1591,E2 84.6077} C_DIS
LIN {X 97.9699,Y 7.9609,Z 100,A -1.3934,B 24.9304,C -1.9267,E1 25.1596,E2 86.8299} C_DIS
LIN {X 98.2498,Y 2.9056,Z 100,A -3.8008,B 24.9296,C -1.9384,E1 25.1598,E2 89.1955} C_DIS
LIN {X 98.2666,Y -2.3222,Z 100,A -7.1594,B 24.9312,C -1.9164,E1 25.1596,E2 92.5859} C_DIS
LIN {X 98.0706,Y -6.604,Z 100,A -9.0668,B 24.9301,C -1.9314,E1 25.1593,E2 94.4465} C_DIS
LIN {X 97.7923,Y -9.9113,Z 100,A -10.8803,B 24.9301,C -1.9299,E1 25.1588,E2 96.2528} C_DIS
LIN {X 97.3762,Y -13.3986,Z 100,A -12.8572,B 24.9304,C -1.9261,E1 25.1581,E2 98.2271} C_DIS
LIN {X 96.5952,Y -18.1927,Z 100,A -15.6189,B 24.9309,C -1.9198,E1 25.1568,E2 100.9875} C_DIS
LIN {X 95.8023,Y -21.9863,Z 100,A -17.5664,B 24.9305,C -1.9249,E1 25.1557,E2 102.9117} C_DIS
LIN {X 95.2668,Y -24.2028,Z 100,A -19.2956,B 24.932,C -1.9048,E1 25.1545,E2 104.6782} C_DIS
LIN {X 94.3401,Y -27.5962,Z 100,A -21.3698,B 24.9325,C -1.8974,E1 25.1529,E2 106.758} C_DIS
LIN {X 92.5772,Y -33.0331,Z 100,A -24.5314,B 24.9328,C -1.8937,E1 25.1502,E2 109.9105} C_DIS
LIN {X 91.4703,Y -35.981,Z 100,A -26.6773,B 24.934,C -1.8758,E1 25.148,E2 112.0866} C_DIS
LIN {X 90.2134,Y -39.0266,Z 100,A -28.4011,B 24.934,C -1.8777,E1 25.1461,E2 113.7966} C_DIS
LIN {X 88.8249,Y -42.0936,Z 100,A -30.2689,B 24.934,C -1.8754,E1 25.1439,E2 115.6596} C_DIS
LIN {X 86.7798,Y -46.1615,Z 100,A -33.4791,B 24.9361,C -1.8459,E1 25.1397,E2 118.9226} C_DIS
LIN {X 84.9535,Y -49.4416,Z 100,A -35.2648,B 24.9355,C -1.8552,E1 25.1373,E2 120.6771} C_DIS
LIN {X 83.2532,Y -52.2533,Z 100,A -37.067,B 24.9355,C -1.8541,E1 25.1346,E2 122.4726} C_DIS
LIN {X 80.0392,Y -57.0543,Z 100,A -40.3207,B 24.9359,C -1.8492,E1 25.1295,E2 125.7219} C_DIS
LIN {X 77.9042,Y -59.9367,Z 100,A -42.4064,B 24.9363,C -1.8437,E1 25.126,E2 127.8105} C_DIS
LIN {X 75.6641,Y -62.7409,Z 100,A -44.4796,B 24.9366,C -1.8389,E1 25.1224,E2 129.8855} C_DIS
LIN {X 73.3244,Y -65.46,Z 100,A -46.5728,B 24.937,C -1.8335,E1 25.1185,E2 131.9821} C_DIS
LIN {X 70.9022,Y -68.0762,Z 100,A -48.6453,B 24.9373,C -1.8285,E1 25.1145,E2 134.0573} C_DIS
LIN {X 68.498,Y -70.4957,Z 100,A -50.6014,B 24.9376,C -1.8249,E1 25.1107,E2 136.0137} C_DIS
LIN {X 66.1818,Y -72.6743,Z 100,A -52.5606,B 24.9382,C -1.8164,E1 25.1066,E2 137.9849} C_DIS
LIN {X 63.4691,Y -75.055,Z 100,A -54.6194,B 24.9384,C -1.8134,E1 25.1023,E2 140.0429} C_DIS
LIN {X 60.8764,Y -77.1721,Z 100,A -56.5592,B 24.9386,C -1.8095,E1 25.098,E2 141.9844} C_DIS
LIN {X 57.1613,Y -79.9628,Z 100,A -59.5672,B 24.9398,C -1.7924,E1 25.0912,E2 145.0222} C_DIS
LIN {X 52.521,Y -83.0859,Z 100,A -62.286,B 24.9388,C -1.8067,E1 25.0849,E2 147.6983} C_DIS
LIN {X 48.2847,Y -85.6166,Z 100,A -65.0878,B 24.939,C -1.8043,E1 25.0782,E2 150.4972} C_DIS
LIN {X 46.4889,Y -86.605,Z 100,A -66.3783,B 24.9394,C -1.7985,E1 25.075,E2 151.7976} C_DIS
LIN {X 43.821,Y -87.9841,Z 100,A -68.2887,B 24.94,C -1.7896,E1 25.0702,E2 153.724} C_DIS
LIN {X 40.3589,Y -89.6249,Z 100,A -70.4444,B 24.94,C -1.789,E1 25.0648,E2 155.8755} C_DIS
LIN {X 34.7782,Y -91.9344,Z 100,A -73.9799,B 24.9404,C -1.7834,E1 25.0556,E2 159.4161} C_DIS
LIN {X 31.389,Y -93.1461,Z 100,A -76.4454,B 24.9415,C -1.767,E1 25.049,E2 161.9156} C_DIS
LIN {X 27.2718,Y -94.4349,Z 100,A -78.5446,B 24.9406,C -1.7796,E1 25.0435,E2 163.9813} C_DIS
LIN {X 24.0054,Y -95.3175,Z 100,A -80.4943,B 24.9407,C -1.7784,E1 25.0382,E2 165.9308} C_DIS
LIN {X 19.6731,Y -96.3039,Z 100,A -82.9702,B 24.9406,C -1.7803,E1 25.0315,E2 168.399} C_DIS
LIN {X 14.8442,Y -97.1655,Z 100,A -85.9126,B 24.941,C -1.7749,E1 25.0234,E2 171.3509} C_DIS
LIN {X 11.5338,Y -97.6137,Z 100,A -88.5867,B 24.9428,C -1.7471,E1 25.0158,E2 174.0889} C_DIS
LIN {X 7.4408,Y -98.0114,Z 100,A -90.1878,B 24.941,C -1.775,E1 25.0115,E2 175.6232} C_DIS
LIN {X 3.0675,Y -98.2448,Z 100,A -92.8882,B 24.9414,C -1.7686,E1 25.004,E2 178.3378} C_DIS
LIN {X 0.7031,Y -98.2806,Z 100,A -94.8963,B 24.9429,C -1.7456,E1 24.9982,E2 180.4003} C_DIS
Enddeposition()
LIN {X 0.7031,Y -98.2806,Z 100,A -94.8963,B 24.9429,C -1.7456,E1 24.9982,E2 180.4003} C_DIS
Startdeposition()
$VEL.CP = VEL_PRINT
LIN {X 2.3662,Y -97.3877,Z 100,A -92.3362,B 24.938,C -1.8186,E1 25.0059,E2 177.6673} C_DIS
LIN {X 6.0828,Y -97.2259,Z 100,A -89.867,B 24.9372,C -1.8299,E1 25.0128,E2 175.1722} C_DIS
LIN {X 11.2953,Y -96.7577,Z 100,A -87.2335,B 24.9382,C -1.8151,E1 25.02,E2 172.5755} C_DIS
LIN {X 14.5931,Y -96.316,Z 100,A -85.1174,B 24.9377,C -1.8224,E1 25.0259,E2 170.444} C_DIS
LIN {X 18.8716,Y -95.5705,Z 100,A -82.666,B 24.9379,C -1.8206,E1 25.0326,E2 167.9997} C_DIS
LIN {X 22.4997,Y -94.7826,Z 100,A -80.5398,B 24.9379,C -1.8205,E1 25.0384,E2 165.8766} C_DIS
LIN {X 25.5063,Y -94.0164,Z 100,A -78.6278,B 24.9375,C -1.8257,E1 25.0436,E2 163.9553} C_DIS
LIN {X 28.2537,Y -93.2293,Z 100,A -76.9162,B 24.9373,C -1.8287,E1 25.0482,E2 162.2395} C_DIS
LIN {X 31.3954,Y -92.2174,Z 100,A -74.9784,B 24.9372,C -1.831,E1 25.0533,E2 160.3} C_DIS
LIN {X 34.8153,Y -90.9816,Z 100,A -72.7203,B 24.9366,C -1.8384,E1 25.0592,E2 158.0291} C_DIS
LIN {X 38.3497,Y -89.5503,Z 100,A -70.5846,B 24.9367,C -1.8376,E1 25.0647,E2 155.9004} C_DIS
LIN {X 41.6719,Y -88.0535,Z 100,A -68.4217,B 24.9364,C -1.8417,E1 25.0702,E2 153.7334} C_DIS
LIN {X 45.0198,Y -86.3889,Z 100,A -66.3107,B 24.9364,C -1.842,E1 25.0754,E2 151.6274} C_DIS
LIN {X 47.9999,Y -84.7702,Z 100,A -64.4914,B 24.9366,C -1.8388,E1 25.0799,E2 149.821} C_DIS
LIN {X 51.1517,Y -82.9062,Z 100,A -61.7396,B 24.9347,C -1.8659,E1 25.0866,E2 147.0137} C_DIS
LIN {X 53.9186,Y -81.1313,Z 100,A -60.124,B 24.9353,C -1.8574,E1 25.0903,E2 145.4235} C_DIS
LIN {X 59.1251,Y -77.4212,Z 100,A -56.4725,B 24.9351,C -1.861,E1 25.0985,E2 141.7765} C_DIS
LIN {X 62.0144,Y -75.1263,Z 100,A -54.4198,B 24.9351,C -1.8612,E1 25.1029,E2 139.7311} C_DIS
LIN {X 64.6107,Y -72.9063,Z 100,A -52.365,B 24.9346,C -1.8676,E1 25.1073,E2 137.6692} C_DIS
LIN {X 67.2131,Y -70.5147,Z 100,A -50.2348,B 24.9341,C -1.8745,E1 25.1116,E2 135.5315} C_DIS
LIN {X 69.7924,Y -67.9625,Z 100,A -48.1634,B 24.9339,C -1.8773,E1 25.1157,E2 133.4624} C_DIS
LIN {X 72.236,Y -65.3595,Z 100,A -46.0654,B 24.9336,C -1.8825,E1 25.1197,E2 131.3612} C_DIS
LIN {X 74.5705,Y -62.6832,Z 100,A -43.9365,B 24.9331,C -1.8895,E1 25.1235,E2 129.2255} C_DIS
LIN {X 76.8989,Y -59.803,Z 100,A -41.8903,B 24.9331,C -1.8901,E1 25.1271,E2 127.1874} C_DIS
LIN {X 78.4462,Y -57.7572,Z 100,A -40.5699,B 24.9333,C -1.8868,E1 25.1293,E2 125.881} C_DIS
LIN {X 82.435,Y -51.906,Z 100,A -36.1773,B 24.9318,C -1.9074,E1 25.1361,E2 121.4617} C_DIS
LIN {X 85.0688,Y -47.4652,Z 100,A -32.8508,B 24.9303,C -1.9276,E1 25.1408,E2 118.1046} C_DIS
LIN {X 87.2077,Y -43.4107,Z 100,A -30.7121,B 24.9314,C -1.9136,E1 25.1435,E2 116.0103} C_DIS
LIN {X 88.8196,Y -40.0089,Z 100,A -28.3096,B 24.9303,C -1.9277,E1 25.1463,E2 113.5876} C_DIS
LIN {X 90.2695,Y -36.6206,Z 100,A -26.0905,B 24.9297,C -1.9364,E1 25.1487,E2 111.3602} C_DIS
LIN {X 91.4366,Y -33.6012,Z 100,A -24.529,B 24.9303,C -1.9287,E1 25.1502,E2 109.8254} C_DIS
LIN {X 92.414,Y -30.8124,Z 100,A -22.5908,B 24.9293,C -1.942,E1 25.152,E2 107.8668} C_DIS
LIN {X 93.2129,Y -28.3077,Z 100,A -20.8543,B 24.9284,C -1.9544,E1 25.1535,E2 106.1109} C_DIS
LIN {X 94.226,Y -24.7254,Z 100,A -19.0253,B 24.9289,C -1.9471,E1 25.1548,E2 104.3098} C_DIS
LIN {X 94.9148,Y -21.9278,Z 100,A -17.3672,B 24.9286,C -1.951,E1 25.1559,E2 102.6518} C_DIS
LIN {X 95.5534,Y -18.96,Z 100,A -15.537,B 24.9281,C -1.9585,E1 25.1569,E2 100.8147} C_DIS
LIN {X 96.1089,Y -15.898,Z 100,A -13.6888,B 24.9276,C -1.9651,E1 25.1578,E2 98.9618} C_DIS
LIN {X 96.5659,Y -12.8361,Z 100,A -12.0351,B 24.9276,C -1.9643,E1 25.1585,E2 97.3196} C_DIS
LIN {X 96.8812,Y -10.1822,Z 100,A -10.2292,B 24.9266,C -1.9787,E1 25.159,E2 95.4906} C_DIS
LIN {X 97.1753,Y -6.8319,Z 100,A -8.3772,B 24.9265,C -1.9801,E1 25.1595,E2 93.6463} C_DIS
LIN {X 97.3564,Y -3.3981,Z 100,A -6.1921,B 24.9255,C -1.993,E1 25.1597,E2 91.4436} C_DIS
LIN {X 97.4155,Y 0.1709,Z 100,A -4.1085,B 24.9251,C -1.9992,E1 25.1597,E2 89.3579} C_DIS
LIN {X 97.322,Y 4.2516,Z 100,A -1.3909,B 24.9235,C -2.0195,E1 25.1595,E2 86.6086} C_DIS
LIN {X 96.9865,Y 9.1267,Z 100,A 0.877,B 24.9247,C -2.0046,E1 25.159,E2 84.3891} C_DIS
LIN {X 96.4845,Y 13.4331,Z 100,A 3.6212,B 24.9235,C -2.0203,E1 25.1581,E2 81.6241} C_DIS
LIN {X 96.126,Y 15.796,Z 100,A 5.0646,B 24.923,C -2.0263,E1 25.1574,E2 80.1752} C_DIS
LIN {X 95.4897,Y 19.2732,Z 100,A 6.8319,B 24.9235,C -2.0205,E1 25.1565,E2 78.432} C_DIS
LIN {X 94.9117,Y 21.9411,Z 100,A 8.7007,B 24.9223,C -2.0358,E1 25.1554,E2 76.5378} C_DIS
LIN {X 94.2475,Y 24.6418,Z 100,A 10.4761,B 24.9215,C -2.0463,E1 25.1541,E2 74.7478} C_DIS
LIN {X 93.1227,Y 28.5986,Z 100,A 12.6441,B 24.9217,C -2.0437,E1 25.1524,E2 72.5982} C_DIS
LIN {X 92.2301,Y 31.3578,Z 100,A 14.2699,B 24.9215,C -2.0457,E1 25.151,E2 70.977} C_DIS
LIN {X 90.8927,Y 35.0499,Z 100,A 16.793,B 24.9204,C -2.0609,E1 25.1485,E2 68.4322} C_DIS
LIN {X 87.9849,Y 41.8144,Z 100,A 20.966,B 24.9199,C -2.067,E1 25.1438,E2 64.2674} C_DIS
LIN {X 86.4932,Y 44.8204,Z 100,A 23.058,B 24.9191,C -2.0771,E1 25.1412,E2 62.1627} C_DIS
LIN {X 84.7167,Y 48.0935,Z 100,A 25.2194,B 24.9187,C -2.0819,E1 25.1382,E2 60.0012} C_DIS
LIN {X 82.8832,Y 51.1885,Z 100,A 27.4013,B 24.9181,C -2.0901,E1 25.1351,E2 57.8112} C_DIS
LIN {X 80.6689,Y 54.6093,Z 100,A 29.5206,B 24.9184,C -2.0855,E1 25.1318,E2 55.7133} C_DIS
LIN {X 78.84,Y 57.2195,Z 100,A 31.3077,B 24.9184,C -2.0868,E1 25.1289,E2 53.9317} C_DIS
LIN {X 77.0535,Y 59.6022,Z 100,A 33.1679,B 24.9177,C -2.0953,E1 25.1258,E2 52.0604} C_DIS
LIN {X 75.1835,Y 61.9455,Z 100,A 35.1077,B 24.9168,C -2.1063,E1 25.1223,E2 50.1037} C_DIS
LIN {X 69.6309,Y 68.1278,Z 100,A 39.9065,B 24.9162,C -2.1137,E1 25.1133,E2 45.3085} C_DIS
LIN {X 67.2075,Y 70.5202,Z 100,A 41.9739,B 24.9157,C -2.1203,E1 25.1091,E2 43.234} C_DIS
LIN {X 64.321,Y 73.1611,Z 100,A 44.3892,B 24.915,C -2.1293,E1 25.1041,E2 40.8071} C_DIS
LIN {X 61.9707,Y 75.1626,Z 100,A 46.4773,B 24.9139,C -2.1431,E1 25.0995,E2 38.6943} C_DIS
LIN {X 59.1474,Y 77.404,Z 100,A 48.6036,B 24.9135,C -2.1472,E1 25.0948,E2 36.5662} C_DIS
LIN {X 56.1859,Y 79.5803,Z 100,A 50.0893,B 24.9153,C -2.1252,E1 25.0916,E2 35.1377} C_DIS
LIN {X 54.443,Y 80.7814,Z 100,A 51.4732,B 24.9147,C -2.1325,E1 25.0883,E2 33.7411} C_DIS
LIN {X 51.2856,Y 82.8226,Z 100,A 53.5934,B 24.9147,C -2.1325,E1 25.0833,E2 31.6277} C_DIS
LIN {X 48.9983,Y 84.1967,Z 100,A 55.3034,B 24.9141,C -2.1401,E1 25.0792,E2 29.9052} C_DIS
LIN {X 46.015,Y 85.8633,Z 100,A 57.287,B 24.914,C -2.1418,E1 25.0743,E2 27.923} C_DIS
LIN {X 42.8373,Y 87.4919,Z 100,A 59.2395,B 24.9142,C -2.139,E1 25.0695,E2 25.9826} C_DIS
LIN {X 40.1322,Y 88.7641,Z 100,A 60.9016,B 24.9143,C -2.1375,E1 25.0653,E2 24.3282} C_DIS
LIN {X 37.5283,Y 89.8965,Z 100,A 62.6757,B 24.9139,C -2.1432,E1 25.0607,E2 22.545} C_DIS
LIN {X 33.8205,Y 91.3566,Z 100,A 65.1494,B 24.9133,C -2.1502,E1 25.0542,E2 20.06} C_DIS
LIN {X 28.0946,Y 93.2765,Z 100,A 68.4904,B 24.9137,C -2.1453,E1 25.0454,E2 16.7369} C_DIS
LIN {X 25.2179,Y 94.0943,Z 100,A 70.2813,B 24.9135,C -2.1477,E1 25.0406,E2 14.9433} C_DIS
LIN {X 22.2515,Y 94.84,Z 100,A 72.185,B 24.9131,C -2.1525,E1 25.0354,E2 13.0309} C_DIS
LIN {X 18.8273,Y 95.579,Z 100,A 74.0456,B 24.9136,C -2.1462,E1 25.0304,E2 11.1877} C_DIS
LIN {X 15.9999,Y 96.0919,Z 100,A 75.9713,B 24.9129,C -2.1553,E1 25.025,E2 9.2423} C_DIS
LIN {X 13.1983,Y 96.5179,Z 100,A 77.4756,B 24.9133,C -2.1499,E1 25.0209,E2 7.7523} C_DIS
LIN {X 10.2548,Y 96.8736,Z 100,A 79.0484,B 24.9138,C -2.1441,E1 25.0166,E2 6.1944} C_DIS
LIN {X 7.0291,Y 97.1619,Z 100,A 81.2685,B 24.9129,C -2.1555,E1 25.0103,E2 3.9484} C_DIS
LIN {X 4.1427,Y 97.3267,Z 100,A 82.935,B 24.9129,C -2.1542,E1 25.0057,E2 2.2854} C_DIS
LIN {X 1.3525,Y 97.4064,Z 100,A 84.9758,B 24.9118,C -2.1683,E1 24.9999,E2 0.2116} C_DIS
LIN {X -3.9001,Y 97.3371,Z 100,A 87.6716,B 24.913,C -2.1533,E1 24.9925,E2 -2.4491} C_DIS
LIN {X -6.9511,Y 97.1672,Z 100,A 89.4126,B 24.9133,C -2.1506,E1 24.9876,E2 -4.1842} C_DIS
LIN {X -9.8217,Y 96.9189,Z 100,A 91.3469,B 24.9126,C -2.1583,E1 24.9822,E2 -6.1377} C_DIS
LIN {X -14.2133,Y 96.3737,Z 100,A 93.8874,B 24.9129,C -2.1544,E1 24.9752,E2 -8.671} C_DIS
LIN {X -18.05,Y 95.7287,Z 100,A 96.047,B 24.9134,C -2.1482,E1 24.9693,E2 -10.818} C_DIS
LIN {X -20.764,Y 95.1761,Z 100,A 97.6515,B 24.9136,C -2.1459,E1 24.9649,E2 -12.4191} C_DIS
LIN {X -24.1749,Y 94.3675,Z 100,A 99.7992,B 24.9136,C -2.147,E1 24.9591,E2 -14.5722} C_DIS
LIN {X -27.0919,Y 93.5734,Z 100,A 101.6892,B 24.9134,C -2.1489,E1 24.954,E2 -16.4699} C_DIS
LIN {X -30.8241,Y 92.4101,Z 100,A 103.5822,B 24.9147,C -2.1322,E1 24.949,E2 -18.3266} C_DIS
LIN {X -35.7798,Y 90.6062,Z 100,A 106.4254,B 24.9158,C -2.1193,E1 24.9417,E2 -21.1448} C_DIS
LIN {X -40.2982,Y 88.6893,Z 100,A 109.7171,B 24.915,C -2.1289,E1 24.9332,E2 -24.4669} C_DIS
LIN {X -44.9547,Y 86.4231,Z 100,A 112.9811,B 24.9148,C -2.1314,E1 24.9249,E2 -27.7456} C_DIS
LIN {X -48.1384,Y 84.6909,Z 100,A 115.3109,B 24.9146,C -2.1344,E1 24.9192,E2 -30.0894} C_DIS
LIN {X -51.6413,Y 82.6003,Z 100,A 117.4311,B 24.9157,C -2.1205,E1 24.9142,E2 -32.183} C_DIS
LIN {X -54.5272,Y 80.7245,Z 100,A 119.4791,B 24.9159,C -2.1174,E1 24.9095,E2 -34.2303} C_DIS
LIN {X -57.4893,Y 78.6424,Z 100,A 121.3408,B 24.917,C -2.1041,E1 24.9053,E2 -36.0668} C_DIS
LIN {X -59.1586,Y 77.3954,Z 100,A 123.1847,B 24.9155,C -2.1223,E1 24.9011,E2 -37.9608} C_DIS
LIN {X -62.6883,Y 74.5662,Z 100,A 125.6566,B 24.9165,C -2.1101,E1 24.8958,E2 -40.4129} C_DIS
LIN {X -65.5213,Y 72.0889,Z 100,A 127.766,B 24.9172,C -2.1016,E1 24.8914,E2 -42.5103} C_DIS
LIN {X -69.7096,Y 68.0481,Z 100,A 131.3015,B 24.9175,C -2.0971,E1 24.8844,E2 -46.05} C_DIS
LIN {X -73.3844,Y 64.0654,Z 100,A 134.4979,B 24.9181,C -2.0894,E1 24.8784,E2 -49.2422} C_DIS
LIN {X -76.7544,Y 59.989,Z 100,A 137.6079,B 24.9188,C -2.0811,E1 24.8729,E2 -52.3471} C_DIS
LIN {X -78.9252,Y 57.103,Z 100,A 139.7134,B 24.9193,C -2.0748,E1 24.8694,E2 -54.4476} C_DIS
LIN {X -81.6993,Y 53.0579,Z 100,A 142.6421,B 24.9198,C -2.0682,E1 24.8649,E2 -57.3752} C_DIS
LIN {X -83.5331,Y 50.1216,Z 100,A 144.7406,B 24.9201,C -2.0644,E1 24.8618,E2 -59.4756} C_DIS
LIN {X -85.3318,Y 46.9942,Z 100,A 146.8378,B 24.9206,C -2.0575,E1 24.859,E2 -61.567} C_DIS
LIN {X -87.1403,Y 43.5466,Z 100,A 149.0127,B 24.9214,C -2.047,E1 24.8562,E2 -63.7285} C_DIS
LIN {X -88.172,Y 41.4181,Z 100,A 150.5218,B 24.9214,C -2.0467,E1 24.8544,E2 -65.2451} C_DIS
LIN {X -90.0879,Y 37.0667,Z 100,A 153.3684,B 24.922,C -2.0398,E1 24.8513,E2 -68.0911} C_DIS
LIN {X -91.3374,Y 33.8732,Z 100,A 155.3558,B 24.9225,C -2.0326,E1 24.8493,E2 -70.0726} C_DIS
LIN {X -92.3609,Y 30.9699,Z 100,A 157.5567,B 24.922,C -2.0398,E1 24.8473,E2 -72.3033} C_DIS
LIN {X -93.8377,Y 26.1592,Z 100,A 160.9024,B 24.9217,C -2.0432,E1 24.8447,E2 -75.6765} C_DIS
LIN {X -94.9329,Y 21.8493,Z 100,A 162.631,B 24.9246,C -2.0058,E1 24.8437,E2 -77.3257} C_DIS
LIN {X -95.3913,Y 19.7529,Z 100,A 165.1711,B 24.9217,C -2.0439,E1 24.8422,E2 -79.9718} C_DIS
LIN {X -96.4023,Y 14.0117,Z 100,A 167.3381,B 24.9257,C -1.9912,E1 24.8413,E2 -82.026} C_DIS
LIN {X -96.7023,Y 11.7682,Z 100,A 168.9091,B 24.9254,C -1.9947,E1 24.8408,E2 -83.6148} C_DIS
LIN {X -97.0677,Y 8.2294,Z 100,A 171.0108,B 24.9259,C -1.9883,E1 24.8402,E2 -85.7138} C_DIS
LIN {X -97.312,Y 4.4832,Z 100,A 172.9795,B 24.927,C -1.9734,E1 24.8399,E2 -87.6587} C_DIS
LIN {X -97.4025,Y 1.5655,Z 100,A 174.9649,B 24.9267,C -1.9766,E1 24.8398,E2 -89.6638} C_DIS
LIN {X -97.4068,Y -1.3277,Z 100,A 176.4065,B 24.9278,C -1.9627,E1 24.8398,E2 -91.0808} C_DIS
LIN {X -97.3244,Y -4.1961,Z 100,A 178.37,B 24.9275,C -1.9663,E1 24.84,E2 -93.0647} C_DIS
LIN {X -97.1562,Y -7.1137,Z 100,A -179.8376,B 24.9277,C -1.9632,E1 24.8404,E2 -94.8605} C_DIS
LIN {X -96.8098,Y -10.8502,Z 100,A -177.7669,B 24.9286,C -1.9517,E1 24.8409,E2 -96.9162} C_DIS
LIN {X -96.3708,Y -14.234,Z 100,A -175.6457,B 24.9288,C -1.9491,E1 24.8418,E2 -99.0439} C_DIS
LIN {X -95.7708,Y -17.8311,Z 100,A -173.6485,B 24.9296,C -1.9375,E1 24.8427,E2 -101.0253} C_DIS
LIN {X -95.1539,Y -20.8661,Z 100,A -171.7109,B 24.9298,C -1.9357,E1 24.8438,E2 -102.97} C_DIS
LIN {X -94.3557,Y -24.2208,Z 100,A -169.8733,B 24.9307,C -1.9232,E1 24.8451,E2 -104.7886} C_DIS
LIN {X -93.3117,Y -27.9757,Z 100,A -167.5641,B 24.9311,C -1.9168,E1 24.8468,E2 -107.0958} C_DIS
LIN {X -91.8935,Y -32.33,Z 100,A -164.71,B 24.9313,C -1.914,E1 24.8494,E2 -109.9596} C_DIS
LIN {X -90.6856,Y -35.5775,Z 100,A -162.6306,B 24.9316,C -1.9095,E1 24.8514,E2 -112.0398} C_DIS
LIN {X -89.7343,Y -37.9131,Z 100,A -160.9676,B 24.9316,C -1.9111,E1 24.8532,E2 -113.7161} C_DIS
LIN {X -88.0578,Y -41.663,Z 100,A -158.7403,B 24.9325,C -1.898,E1 24.8558,E2 -115.9242} C_DIS
LIN {X -87.0184,Y -43.7925,Z 100,A -157.1816,B 24.9324,C -1.8996,E1 24.8578,E2 -117.4951} C_DIS
LIN {X -85.2303,Y -47.176,Z 100,A -155.0113,B 24.933,C -1.8908,E1 24.8606,E2 -119.6559} C_DIS
LIN {X -81.8083,Y -52.888,Z 100,A -150.9742,B 24.9334,C -1.8845,E1 24.8665,E2 -123.6987} C_DIS
LIN {X -79.5573,Y -56.2181,Z 100,A -148.9165,B 24.9346,C -1.8683,E1 24.8697,E2 -125.7278} C_DIS
LIN {X -78.4002,Y -57.8201,Z 100,A -147.2664,B 24.9336,C -1.8818,E1 24.8725,E2 -127.4183} C_DIS
LIN {X -75.8322,Y -61.1488,Z 100,A -145.0345,B 24.9346,C -1.8678,E1 24.8764,E2 -129.6271} C_DIS
LIN {X -73.4713,Y -63.9658,Z 100,A -143.0115,B 24.9353,C -1.8581,E1 24.88,E2 -131.6364} C_DIS
LIN {X -70.4918,Y -67.2369,Z 100,A -140.4387,B 24.9358,C -1.8513,E1 24.8849,E2 -134.2042} C_DIS
LIN {X -67.2058,Y -70.5218,Z 100,A -137.4115,B 24.9355,C -1.8556,E1 24.8909,E2 -137.2544} C_DIS
LIN {X -64.545,Y -72.9652,Z 100,A -135.3295,B 24.9359,C -1.8499,E1 24.8952,E2 -139.3311} C_DIS
LIN {X -62.1444,Y -75.0182,Z 100,A -132.8963,B 24.9347,C -1.8663,E1 24.9006,E2 -141.8127} C_DIS
LIN {X -58.9885,Y -77.5264,Z 100,A -131.1814,B 24.9366,C -1.8393,E1 24.9042,E2 -143.4696} C_DIS
LIN {X -56.416,Y -79.4161,Z 100,A -129.3162,B 24.9368,C -1.8357,E1 24.9085,E2 -145.3327} C_DIS
LIN {X -53.1689,Y -81.6272,Z 100,A -126.8162,B 24.9366,C -1.8386,E1 24.9143,E2 -147.8478} C_DIS
LIN {X -50.3934,Y -83.3678,Z 100,A -125.0979,B 24.9373,C -1.8285,E1 24.9183,E2 -149.5475} C_DIS
LIN {X -47.4882,Y -85.0559,Z 100,A -123.0012,B 24.9373,C -1.8299,E1 24.9234,E2 -151.6537} C_DIS
LIN {X -44.1903,Y -86.8152,Z 100,A -120.9429,B 24.9378,C -1.8222,E1 24.9285,E2 -153.6992} C_DIS
LIN {X -41.3763,Y -88.1914,Z 100,A -119.2576,B 24.9383,C -1.8145,E1 24.9327,E2 -155.3706} C_DIS
LIN {X -39.1119,Y -89.2185,Z 100,A -117.3812,B 24.9374,C -1.8274,E1 24.9376,E2 -157.2823} C_DIS
LIN {X -35.6283,Y -90.6657,Z 100,A -115.528,B 24.9384,C -1.8123,E1 24.9423,E2 -159.1037} C_DIS
LIN {X -31.4552,Y -92.1972,Z 100,A -112.6367,B 24.9379,C -1.8198,E1 24.95,E2 -162.0185} C_DIS
LIN {X -28.0034,Y -93.3035,Z 100,A -110.5426,B 24.9381,C -1.8168,E1 24.9555,E2 -164.1093} C_DIS
LIN {X -24.7493,Y -94.2199,Z 100,A -108.4291,B 24.9379,C -1.8201,E1 24.9613,E2 -166.2338} C_DIS
LIN {X -21.2862,Y -95.0622,Z 100,A -106.3157,B 24.9379,C -1.8196,E1 24.967,E2 -168.3489} C_DIS
LIN {X -17.5319,Y -95.8246,Z 100,A -104.4589,B 24.939,C -1.8045,E1 24.972,E2 -170.1719} C_DIS
LIN {X -15.1453,Y -96.2306,Z 100,A -102.655,B 24.9381,C -1.8178,E1 24.9771,E2 -172.0089} C_DIS
LIN {X -12.3789,Y -96.6252,Z 100,A -100.7462,B 24.9374,C -1.8272,E1 24.9824,E2 -173.9414} C_DIS
LIN {X -7.2535,Y -97.1457,Z 100,A -97.3126,B 24.9364,C -1.8419,E1 24.9921,E2 -177.4114} C_DIS
LIN {X -2.8268,Y -97.3739,Z 100,A -94.9493,B 24.937,C -1.8332,E1 24.9986,E2 -179.7545} C_DIS
LIN {X 0.7124,Y -97.4115,Z 100,A -94.7848,B 24.9417,C -1.7638,E1 24.9986,E2 -179.7545} C_DIS
Enddeposition()
LIN {X 0.7124,Y -97.4115,Z 100,A -94.7848,B 24.9417,C -1.7638,E1 24.9986,E2 -179.7545} C_DIS
Startdeposition()
$VEL.CP = VEL_PRINT
LIN {X -0.105,Y -96.538,Z 100,A -94.7217,B 24.9394,C -1.7988,E1 24.999,E2 -179.9006} C_DIS
LIN {X -2.4331,Y -96.5076,Z 100,A -96.1086,B 24.9394,C -1.7984,E1 24.9952,E2 -178.5125} C_DIS
LIN {X -4.7741,Y -96.4203,Z 100,A -97.5016,B 24.9394,C -1.7982,E1 24.9913,E2 -177.1187} C_DIS
LIN {X -7.1181,Y -96.2758,Z 100,A -98.8374,B 24.9393,C -1.8002,E1 24.9876,E2 -175.7873} C_DIS
LIN {X -9.5793,Y -96.0616,Z 100,A -100.2553,B 24.9391,C -1.802,E1 24.9836,E2 -174.3729} C_DIS
LIN {X -11.8303,Y -95.811,Z 100,A -101.6512,B 24.9392,C -1.8004,E1 24.9797,E2 -172.9723} C_DIS
LIN {X -14.2879,Y -95.4748,Z 100,A -103.0668,B 24.9391,C -1.8027,E1 24.9758,E2 -171.561} C_DIS
LIN {X -16.5149,Y -95.1155,Z 100,A -104.6524,B 24.9396,C -1.7944,E1 24.9714,E2 -169.9543} C_DIS
LIN {X -18.9567,Y -94.6585,Z 100,A -105.9406,B 24.9392,C -1.8016,E1 24.9679,E2 -168.6815} C_DIS
LIN {X -21.1511,Y -94.1931,Z 100,A -107.2747,B 24.9392,C -1.8021,E1 24.9643,E2 -167.3469} C_DIS
LIN {X -23.5857,Y -93.6125,Z 100,A -108.7609,B 24.9391,C -1.8028,E1 24.9602,E2 -165.8605} C_DIS
LIN {X -25.7557,Y -93.0395,Z 100,A -110.2758,B 24.9395,C -1.7973,E1 24.9561,E2 -164.3302} C_DIS
LIN {X -29.2738,Y -91.9925,Z 100,A -112.2097,B 24.9388,C -1.8074,E1 24.951,E2 -162.4168} C_DIS
LIN {X -31.4408,Y -91.2751,Z 100,A -113.6888,B 24.939,C -1.8042,E1 24.9471,E2 -160.9273} C_DIS
LIN {X -33.7666,Y -90.44,Z 100,A -115.1009,B 24.9388,C -1.8074,E1 24.9434,E2 -159.52} C_DIS
LIN {X -35.9611,Y -89.5901,Z 100,A -116.6533,B 24.939,C -1.8033,E1 24.9393,E2 -157.9547} C_DIS
LIN {X -39.1335,Y -88.2512,Z 100,A -118.5514,B 24.9386,C -1.8105,E1 24.9345,E2 -156.0691} C_DIS
LIN {X -41.2831,Y -87.2663,Z 100,A -120.0184,B 24.9386,C -1.8099,E1 24.9308,E2 -154.5971} C_DIS
LIN {X -43.6141,Y -86.1238,Z 100,A -121.4495,B 24.9382,C -1.8156,E1 24.9272,E2 -153.1757} C_DIS
LIN {X -45.6133,Y -85.0824,Z 100,A -122.7807,B 24.9381,C -1.8175,E1 24.9239,E2 -151.8455} C_DIS
LIN {X -47.579,Y -83.9997,Z 100,A -124.1824,B 24.9381,C -1.817,E1 24.9205,E2 -150.4384} C_DIS
LIN {X -49.6342,Y -82.8019,Z 100,A -125.818,B 24.9385,C -1.8114,E1 24.9165,E2 -148.7846} C_DIS
LIN {X -52.6526,Y -80.9161,Z 100,A -127.7157,B 24.9378,C -1.8219,E1 24.9121,E2 -146.9058} C_DIS
LIN {X -54.7145,Y -79.5356,Z 100,A -129.1757,B 24.9376,C -1.8248,E1 24.9087,E2 -145.4477} C_DIS
LIN {X -56.5545,Y -78.2388,Z 100,A -130.7327,B 24.9379,C -1.8196,E1 24.9051,E2 -143.8728} C_DIS
LIN {X -58.9519,Y -76.4463,Z 100,A -132.4603,B 24.9376,C -1.8244,E1 24.9013,E2 -142.1505} C_DIS
LIN {X -61.7566,Y -74.199,Z 100,A -134.5526,B 24.9372,C -1.8297,E1 24.8968,E2 -140.063} C_DIS
LIN {X -64.3883,Y -71.9271,Z 100,A -136.6425,B 24.937,C -1.8329,E1 24.8924,E2 -137.9723} C_DIS
LIN {X -66.9797,Y -69.5204,Z 100,A -138.6414,B 24.9365,C -1.8405,E1 24.8884,E2 -135.9834} C_DIS
LIN {X -69.2311,Y -67.2798,Z 100,A -140.4301,B 24.936,C -1.8477,E1 24.8849,E2 -134.2042} C_DIS
LIN {X -70.7907,Y -65.6376,Z 100,A -142.0717,B 24.9365,C -1.8408,E1 24.8817,E2 -132.5389} C_DIS
LIN {X -73.1082,Y -63.0468,Z 100,A -144.1744,B 24.9363,C -1.8441,E1 24.8778,E2 -130.4349} C_DIS
LIN {X -75.3692,Y -60.3258,Z 100,A -146.2874,B 24.9359,C -1.8486,E1 24.8741,E2 -128.3228} C_DIS
LIN {X -77.5429,Y -57.5049,Z 100,A -148.2564,B 24.9353,C -1.8585,E1 24.8708,E2 -126.3678} C_DIS
LIN {X -78.9286,Y -55.5878,Z 100,A -149.7939,B 24.9353,C -1.8576,E1 24.8683,E2 -124.8208} C_DIS
LIN {X -80.9229,Y -52.6421,Z 100,A -151.929,B 24.935,C -1.8623,E1 24.865,E2 -122.6859} C_DIS
LIN {X -82.3839,Y -50.3221,Z 100,A -153.3215,B 24.9342,C -1.8742,E1 24.863,E2 -121.3148} C_DIS
LIN {X -83.5013,Y -48.4464,Z 100,A -154.7455,B 24.9342,C -1.8734,E1 24.8609,E2 -119.8817} C_DIS
LIN {X -85.1427,Y -45.502,Z 100,A -156.6836,B 24.9337,C -1.8809,E1 24.8583,E2 -117.9511} C_DIS
LIN {X -86.232,Y -43.4023,Z 100,A -158.1565,B 24.9336,C -1.8825,E1 24.8565,E2 -116.4743} C_DIS
LIN {X -87.3204,Y -41.1671,Z 100,A -159.7274,B 24.9335,C -1.8836,E1 24.8546,E2 -114.8973} C_DIS
LIN {X -88.7826,Y -37.9107,Z 100,A -161.6462,B 24.9326,C -1.8961,E1 24.8524,E2 -112.9978} C_DIS
LIN {X -89.7127,Y -35.6532,Z 100,A -163.0609,B 24.9322,C -1.9014,E1 24.8509,E2 -111.5879} C_DIS
LIN {X -90.4899,Y -33.6347,Z 100,A -164.5232,B 24.9324,C -1.8994,E1 24.8495,E2 -110.1125} C_DIS
LIN {X -91.3367,Y -31.2596,Z 100,A -165.8998,B 24.9318,C -1.9077,E1 24.8482,E2 -108.7479} C_DIS
LIN {X -92.0698,Y -29.0299,Z 100,A -167.3192,B 24.9315,C -1.911,E1 24.847,E2 -107.3284} C_DIS
LIN {X -92.7487,Y -26.7819,Z 100,A -168.9306,B 24.9317,C -1.9083,E1 24.8457,E2 -105.701} C_DIS
LIN {X -93.6142,Y -23.5787,Z 100,A -170.9574,B 24.9314,C -1.9124,E1 24.8443,E2 -103.6724} C_DIS
LIN {X -94.1943,Y -21.146,Z 100,A -172.252,B 24.9307,C -1.9231,E1 24.8435,E2 -102.3955} C_DIS
LIN {X -94.7069,Y -18.7133,Z 100,A -173.7376,B 24.9304,C -1.9273,E1 24.8427,E2 -100.9114} C_DIS
LIN {X -95.137,Y -16.3873,Z 100,A -175.0867,B 24.9299,C -1.9335,E1 24.842,E2 -99.5689} C_DIS
LIN {X -95.5101,Y -14.0506,Z 100,A -176.6022,B 24.9299,C -1.9343,E1 24.8413,E2 -98.0464} C_DIS
LIN {X -95.828,Y -11.686,Z 100,A -178.1291,B 24.9298,C -1.9353,E1 24.8408,E2 -96.5127} C_DIS
LIN {X -96.0855,Y -9.3363,Z 100,A -179.4038,B 24.9292,C -1.9438,E1 24.8405,E2 -95.2507} C_DIS
LIN {X -96.2771,Y -7.1013,Z 100,A 179.195,B 24.929,C -1.9458,E1 24.8401,E2 -93.8459} C_DIS
LIN {X -96.4221,Y -4.7418,Z 100,A 177.6474,B 24.929,C -1.9458,E1 24.8399,E2 -92.2887} C_DIS
LIN {X -96.5335,Y -0.8552,Z 100,A 175.6822,B 24.9277,C -1.964,E1 24.8398,E2 -90.3553} C_DIS
LIN {X -96.5291,Y 1.3093,Z 100,A 174.291,B 24.9277,C -1.9648,E1 24.8398,E2 -88.9575} C_DIS
LIN {X -96.4681,Y 3.6731,Z 100,A 172.876,B 24.9273,C -1.9689,E1 24.8399,E2 -87.5438} C_DIS
LIN {X -96.3492,Y 6.0346,Z 100,A 171.4601,B 24.927,C -1.973,E1 24.8401,E2 -86.1293} C_DIS
LIN {X -96.1591,Y 8.5389,Z 100,A 169.9592,B 24.9267,C -1.9775,E1 24.8405,E2 -84.63} C_DIS
LIN {X -95.9501,Y 10.6437,Z 100,A 168.5331,B 24.9267,C -1.9761,E1 24.8409,E2 -83.1921} C_DIS
LIN {X -95.6604,Y 12.9922,Z 100,A 167.2166,B 24.9262,C -1.9834,E1 24.8414,E2 -81.8851} C_DIS
LIN {X -95.2016,Y 16.0011,Z 100,A 165.2356,B 24.9262,C -1.9837,E1 24.8423,E2 -79.8929} C_DIS
LIN {X -94.6398,Y 19.0478,Z 100,A 163.3845,B 24.9258,C -1.9891,E1 24.8432,E2 -78.044} C_DIS
LIN {X -93.9144,Y 22.3549,Z 100,A 161.4701,B 24.9251,C -1.9985,E1 24.8444,E2 -76.1408} C_DIS
LIN {X -93.3125,Y 24.7455,Z 100,A 160.1194,B 24.9245,C -2.0067,E1 24.8453,E2 -74.8018} C_DIS
LIN {X -92.6828,Y 27.0087,Z 100,A 158.6151,B 24.9245,C -2.0076,E1 24.8465,E2 -73.2909} C_DIS
LIN {X -91.9881,Y 29.2874,Z 100,A 157.2894,B 24.9239,C -2.0149,E1 24.8476,E2 -71.9748} C_DIS
LIN {X -91.2848,Y 31.4131,Z 100,A 155.781,B 24.9239,C -2.0133,E1 24.8489,E2 -70.4539} C_DIS
LIN {X -90.4471,Y 33.7478,Z 100,A 154.3633,B 24.9235,C -2.0195,E1 24.8503,E2 -69.0433} C_DIS
LIN {X -89.5953,Y 35.9484,Z 100,A 153.0515,B 24.923,C -2.0267,E1 24.8516,E2 -67.7411} C_DIS
LIN {X -88.6902,Y 38.1268,Z 100,A 151.6339,B 24.9227,C -2.0304,E1 24.8532,E2 -66.3244} C_DIS
LIN {X -87.769,Y 40.2033,Z 100,A 150.2252,B 24.9225,C -2.0325,E1 24.8548,E2 -64.9131} C_DIS
LIN {X -86.5163,Y 42.8287,Z 100,A 148.6677,B 24.9217,C -2.0431,E1 24.8567,E2 -63.3724} C_DIS
LIN {X -85.6277,Y 44.581,Z 100,A 147.314,B 24.9219,C -2.0405,E1 24.8584,E2 -62.0053} C_DIS
LIN {X -84.5697,Y 46.5583,Z 100,A 145.9746,B 24.9216,C -2.0441,E1 24.8602,E2 -60.6675} C_DIS
LIN {X -83.4046,Y 48.6147,Z 100,A 144.5631,B 24.9214,C -2.0479,E1 24.8621,E2 -59.2575} C_DIS
LIN {X -82.1255,Y 50.7444,Z 100,A 143.0522,B 24.9211,C -2.0509,E1 24.8643,E2 -57.7462} C_DIS
LIN {X -80.8975,Y 52.6807,Z 100,A 141.7124,B 24.9208,C -2.0554,E1 24.8664,E2 -56.4103} C_DIS
LIN {X -79.5204,Y 54.7363,Z 100,A 140.2994,B 24.9203,C -2.0613,E1 24.8686,E2 -55.0043} C_DIS
LIN {X -78.2318,Y 56.564,Z 100,A 138.8385,B 24.9203,C -2.0606,E1 24.8709,E2 -53.5346} C_DIS
LIN {X -76.4673,Y 58.9247,Z 100,A 137.0174,B 24.9202,C -2.063,E1 24.874,E2 -51.7104} C_DIS
LIN {X -74.1642,Y 61.7985,Z 100,A 134.8388,B 24.9197,C -2.0689,E1 24.8779,E2 -49.536} C_DIS
LIN {X -71.8659,Y 64.4567,Z 100,A 132.7197,B 24.9194,C -2.0732,E1 24.8818,E2 -47.4174} C_DIS
LIN {X -69.5048,Y 66.9959,Z 100,A 130.6495,B 24.919,C -2.0778,E1 24.8857,E2 -45.3493} C_DIS
LIN {X -67.3303,Y 69.1825,Z 100,A 128.7556,B 24.9189,C -2.0802,E1 24.8895,E2 -43.453} C_DIS
LIN {X -64.807,Y 71.5523,Z 100,A 126.6577,B 24.9186,C -2.0835,E1 24.8938,E2 -41.3546} C_DIS
LIN {X -62.1478,Y 73.8739,Z 100,A 124.5466,B 24.9183,C -2.0877,E1 24.8983,E2 -39.2452} C_DIS
LIN {X -59.3702,Y 76.124,Z 100,A 122.6306,B 24.9174,C -2.099,E1 24.9024,E2 -37.349} C_DIS
LIN {X -57.3944,Y 77.6238,Z 100,A 121.151,B 24.9172,C -2.1018,E1 24.9057,E2 -35.8709} C_DIS
LIN {X -55.5777,Y 78.9356,Z 100,A 119.7553,B 24.9172,C -2.1023,E1 24.9089,E2 -34.4716} C_DIS
LIN {X -52.6439,Y 80.9218,Z 100,A 117.7022,B 24.9167,C -2.1081,E1 24.9136,E2 -32.4252} C_DIS
LIN {X -50.5453,Y 82.2482,Z 100,A 116.2236,B 24.9165,C -2.1106,E1 24.9171,E2 -30.9482} C_DIS
LIN {X -48.4959,Y 83.4729,Z 100,A 114.8003,B 24.9163,C -2.113,E1 24.9206,E2 -29.5261} C_DIS
LIN {X -46.5425,Y 84.5784,Z 100,A 113.4641,B 24.9161,C -2.1152,E1 24.9238,E2 -28.1913} C_DIS
LIN {X -44.2798,Y 85.7836,Z 100,A 111.962,B 24.9158,C -2.1184,E1 24.9275,E2 -26.6927} C_DIS
LIN {X -42.0979,Y 86.8748,Z 100,A 110.4722,B 24.9158,C -2.1193,E1 24.9313,E2 -25.2011} C_DIS
LIN {X -40.0369,Y 87.8441,Z 100,A 109.197,B 24.9154,C -2.1239,E1 24.9345,E2 -23.9338} C_DIS
LIN {X -37.4835,Y 88.9626,Z 100,A 107.3567,B 24.9157,C -2.1201,E1 24.9392,E2 -22.0801} C_DIS
LIN {X -34.7509,Y 90.0671,Z 100,A 105.7113,B 24.9152,C -2.1259,E1 24.9435,E2 -20.4449} C_DIS
LIN {X -31.9831,Y 91.0848,Z 100,A 103.8373,B 24.9154,C -2.124,E1 24.9484,E2 -18.5627} C_DIS
LIN {X -29.0346,Y 92.0683,Z 100,A 102.1734,B 24.9147,C -2.1323,E1 24.9528,E2 -16.9154} C_DIS
LIN {X -26.7703,Y 92.752,Z 100,A 100.766,B 24.9147,C -2.1337,E1 24.9566,E2 -15.5091} C_DIS
LIN {X -24.6068,Y 93.35,Z 100,A 99.3006,B 24.9149,C -2.1306,E1 24.9605,E2 -14.0338} C_DIS
LIN {X -22.1696,Y 93.9579,Z 100,A 97.7314,B 24.9149,C -2.1293,E1 24.9648,E2 -12.4596} C_DIS
LIN {X -18.9415,Y 94.6616,Z 100,A 95.8365,B 24.9147,C -2.1332,E1 24.97,E2 -10.5717} C_DIS
LIN {X -16.3804,Y 95.1381,Z 100,A 94.424,B 24.9142,C -2.139,E1 24.9738,E2 -9.1714} C_DIS
LIN {X -13.6837,Y 95.5622,Z 100,A 92.8808,B 24.9139,C -2.1427,E1 24.9781,E2 -7.6358} C_DIS
LIN {X -11.667,Y 95.8303,Z 100,A 91.5923,B 24.9141,C -2.1407,E1 24.9816,E2 -6.3414} C_DIS
LIN {X -9.3225,Y 96.0867,Z 100,A 90.1256,B 24.9141,C -2.1391,E1 24.9857,E2 -4.8702} C_DIS
LIN {X -7.0912,Y 96.2778,Z 100,A 88.7355,B 24.9143,C -2.1376,E1 24.9896,E2 -3.4758} C_DIS
LIN {X -4.7351,Y 96.4225,Z 100,A 87.3055,B 24.9143,C -2.1371,E1 24.9936,E2 -2.0442} C_DIS
LIN {X -2.3191,Y 96.5105,Z 100,A 85.9016,B 24.9143,C -2.1386,E1 24.9975,E2 -0.6438} C_DIS
LIN {X 0.0328,Y 96.5385,Z 100,A 84.5032,B 24.9143,C -2.1388,E1 25.0014,E2 0.7541} C_DIS
LIN {X 2.3882,Y 96.509,Z 100,A 83.1037,B 24.9142,C -2.1389,E1 25.0053,E2 2.1532} C_DIS
LIN {X 4.7438,Y 96.422,Z 100,A 81.7037,B 24.9142,C -2.1389,E1 25.0092,E2 3.5527} C_DIS
LIN {X 7.6408,Y 96.234,Z 100,A 79.9281,B 24.9143,C -2.1371,E1 25.0142,E2 5.3318} C_DIS
LIN {X 10.6455,Y 95.9499,Z 100,A 78.2419,B 24.9141,C -2.1405,E1 25.0188,E2 7.0089} C_DIS
LIN {X 13.0032,Y 95.6589,Z 100,A 76.6289,B 24.9147,C -2.133,E1 25.0233,E2 8.6382} C_DIS
LIN {X 16.5075,Y 95.1168,Z 100,A 74.7357,B 24.9141,C -2.1398,E1 25.0285,E2 10.5134} C_DIS
LIN {X 18.95,Y 94.6598,Z 100,A 73.1919,B 24.9144,C -2.1368,E1 25.0328,E2 12.0626} C_DIS
LIN {X 21.1615,Y 94.1907,Z 100,A 71.9216,B 24.9142,C -2.1386,E1 25.0362,E2 13.3269} C_DIS
LIN {X 23.9546,Y 93.5176,Z 100,A 70.3962,B 24.9138,C -2.1441,E1 25.0403,E2 14.8371} C_DIS
LIN {X 27.0061,Y 92.6836,Z 100,A 68.3825,B 24.9143,C -2.1379,E1 25.0458,E2 16.8621} C_DIS
LIN {X 29.3033,Y 91.983,Z 100,A 66.7868,B 24.9149,C -2.1307,E1 25.05,E2 18.4719} C_DIS
LIN {X 32.4166,Y 90.9327,Z 100,A 64.9087,B 24.9148,C -2.1316,E1 25.055,E2 20.3442} C_DIS
LIN {X 34.8736,Y 90.0189,Z 100,A 63.4219,B 24.9148,C -2.1326,E1 25.0589,E2 21.8254} C_DIS
LIN {X 36.9558,Y 89.185,Z 100,A 62.0343,B 24.915,C -2.1292,E1 25.0625,E2 23.218} C_DIS
LIN {X 39.1285,Y 88.2534,Z 100,A 60.694,B 24.915,C -2.1299,E1 25.0659,E2 24.5533} C_DIS
LIN {X 41.2781,Y 87.2688,Z 100,A 59.2343,B 24.9152,C -2.1262,E1 25.0696,E2 26.0181} C_DIS
LIN {X 43.5103,Y 86.1768,Z 100,A 57.8234,B 24.9152,C -2.1267,E1 25.0731,E2 27.424} C_DIS
LIN {X 45.6076,Y 85.0855,Z 100,A 56.4811,B 24.9152,C -2.1271,E1 25.0764,E2 28.7617} C_DIS
LIN {X 47.5884,Y 83.9944,Z 100,A 55.0835,B 24.9155,C -2.1231,E1 25.0798,E2 30.1644} C_DIS
LIN {X 50.1513,Y 82.4877,Z 100,A 53.2213,B 24.9159,C -2.117,E1 25.0843,E2 32.0355} C_DIS
LIN {X 52.8674,Y 80.7744,Z 100,A 51.5681,B 24.9154,C -2.1233,E1 25.0882,E2 33.6684} C_DIS
LIN {X 54.7168,Y 79.534,Z 100,A 50.0369,B 24.9162,C -2.1134,E1 25.0917,E2 35.2179} C_DIS
LIN {X 56.7047,Y 78.1288,Z 100,A 48.6443,B 24.9162,C -2.1128,E1 25.0949,E2 36.6068} C_DIS
LIN {X 58.9743,Y 76.429,Z 100,A 46.8602,B 24.9168,C -2.1061,E1 25.0989,E2 38.4004} C_DIS
LIN {X 61.7007,Y 74.2455,Z 100,A 44.8254,B 24.917,C -2.1036,E1 25.1033,E2 40.4334} C_DIS
LIN {X 64.3911,Y 71.9246,Z 100,A 42.7218,B 24.9173,C -2.0997,E1 25.1077,E2 42.538} C_DIS
LIN {X 66.9907,Y 69.5098,Z 100,A 40.6204,B 24.9176,C -2.0955,E1 25.112,E2 44.6406} C_DIS
LIN {X 69.6324,Y 66.8635,Z 100,A 38.4027,B 24.918,C -2.0908,E1 25.1163,E2 46.86} C_DIS
LIN {X 71.9663,Y 64.3446,Z 100,A 36.4043,B 24.9183,C -2.0877,E1 25.1201,E2 48.8569} C_DIS
LIN {X 74.2519,Y 61.6929,Z 100,A 34.3194,B 24.9187,C -2.0826,E1 25.1238,E2 50.9442} C_DIS
LIN {X 76.4692,Y 58.9222,Z 100,A 32.2255,B 24.919,C -2.078,E1 25.1275,E2 53.0392} C_DIS
LIN {X 78.3214,Y 56.4387,Z 100,A 30.5718,B 24.9188,C -2.0804,E1 25.1302,E2 54.6792} C_DIS
LIN {X 79.9216,Y 54.1471,Z 100,A 28.7386,B 24.9197,C -2.0697,E1 25.1331,E2 56.5289} C_DIS
LIN {X 81.6167,Y 51.5589,Z 100,A 27.02,B 24.9197,C -2.0693,E1 25.1357,E2 58.2396} C_DIS
LIN {X 83.0717,Y 49.1779,Z 100,A 25.5595,B 24.9195,C -2.0724,E1 25.1378,E2 59.6854} C_DIS
LIN {X 84.0604,Y 47.4703,Z 100,A 24.2835,B 24.92,C -2.0652,E1 25.1396,E2 60.9717} C_DIS
LIN {X 85.1414,Y 45.5044,Z 100,A 22.8947,B 24.9205,C -2.0594,E1 25.1414,E2 62.367} C_DIS
LIN {X 86.2303,Y 43.4057,Z 100,A 21.4019,B 24.921,C -2.0521,E1 25.1433,E2 63.8692} C_DIS
LIN {X 87.3497,Y 41.1043,Z 100,A 19.9962,B 24.921,C -2.0521,E1 25.145,E2 65.2672} C_DIS
LIN {X 88.2726,Y 39.0848,Z 100,A 18.6272,B 24.9215,C -2.0464,E1 25.1466,E2 66.6422} C_DIS
LIN {X 89.1967,Y 36.9275,Z 100,A 17.292,B 24.9216,C -2.0446,E1 25.148,E2 67.9744} C_DIS
LIN {X 90.1397,Y 34.5594,Z 100,A 15.8991,B 24.9216,C -2.0448,E1 25.1495,E2 69.3591} C_DIS
LIN {X 90.9378,Y 32.402,Z 100,A 14.4363,B 24.9222,C -2.037,E1 25.1509,E2 70.8321} C_DIS
LIN {X 91.6668,Y 30.2806,Z 100,A 13.0539,B 24.9226,C -2.0311,E1 25.1521,E2 72.2207} C_DIS
LIN {X 92.3812,Y 28.0256,Z 100,A 11.6596,B 24.9229,C -2.0272,E1 25.1532,E2 73.6162} C_DIS
LIN {X 93.0456,Y 25.7336,Z 100,A 10.3125,B 24.9231,C -2.0256,E1 25.1543,E2 74.9594} C_DIS
LIN {X 93.6763,Y 23.331,Z 100,A 8.7254,B 24.9237,C -2.0167,E1 25.1554,E2 76.5583} C_DIS
LIN {X 94.4456,Y 19.9935,Z 100,A 6.7688,B 24.924,C -2.0133,E1 25.1566,E2 78.5114} C_DIS
LIN {X 94.9282,Y 17.5563,Z 100,A 5.3559,B 24.9242,C -2.0111,E1 25.1573,E2 79.9214} C_DIS
LIN {X 95.3135,Y 15.331,Z 100,A 3.8591,B 24.9249,C -2.0009,E1 25.158,E2 81.4335} C_DIS
LIN {X 95.6804,Y 12.8381,Z 100,A 2.5505,B 24.9247,C -2.0034,E1 25.1585,E2 82.7286} C_DIS
LIN {X 95.9523,Y 10.6232,Z 100,A 1.1066,B 24.9254,C -1.9945,E1 25.159,E2 84.1847} C_DIS
LIN {X 96.22,Y 7.8158,Z 100,A -0.3565,B 24.9252,C -1.9974,E1 25.1593,E2 85.6325} C_DIS
LIN {X 96.3663,Y 5.7514,Z 100,A -1.5835,B 24.9255,C -1.9935,E1 25.1595,E2 86.8614} C_DIS
LIN {X 96.4779,Y 3.4017,Z 100,A -2.9699,B 24.9258,C -1.9894,E1 25.1597,E2 88.2493} C_DIS
LIN {X 96.5336,Y 0.848,Z 100,A -4.3804,B 24.9258,C -1.9886,E1 25.1597,E2 89.6532} C_DIS
LIN {X 96.5199,Y -1.8106,Z 100,A -6.2065,B 24.9269,C -1.9739,E1 25.1597,E2 91.5031} C_DIS
LIN {X 96.4212,Y -4.7593,Z 100,A -7.9054,B 24.9272,C -1.9702,E1 25.1595,E2 93.2005} C_DIS
LIN {X 96.2759,Y -7.1165,Z 100,A -9.2387,B 24.9274,C -1.9683,E1 25.1593,E2 94.5304} C_DIS
LIN {X 96.0604,Y -9.5902,Z 100,A -10.6369,B 24.9274,C -1.9665,E1 25.1589,E2 95.9245} C_DIS
LIN {X 95.8125,Y -11.8186,Z 100,A -12.0248,B 24.928,C -1.96,E1 25.1585,E2 97.3197} C_DIS
LIN {X 95.4762,Y -14.2791,Z 100,A -13.4264,B 24.9281,C -1.9581,E1 25.1579,E2 98.7175} C_DIS
LIN {X 94.9074,Y -17.6719,Z 100,A -15.5748,B 24.9289,C -1.9474,E1 25.1569,E2 100.8787} C_DIS
LIN {X 94.4178,Y -20.121,Z 100,A -16.922,B 24.9289,C -1.9479,E1 25.1561,E2 102.2168} C_DIS
LIN {X 93.9145,Y -22.3545,Z 100,A -18.3735,B 24.9294,C -1.9399,E1 25.1552,E2 103.6785} C_DIS
LIN {X 93.3195,Y -24.7198,Z 100,A -19.7109,B 24.9294,C -1.9396,E1 25.1543,E2 105.009} C_DIS
LIN {X 92.6862,Y -26.9976,Z 100,A -21.1071,B 24.9298,C -1.9354,E1 25.1532,E2 106.407} C_DIS
LIN {X 91.9974,Y -29.2589,Z 100,A -22.5034,B 24.9301,C -1.9313,E1 25.1521,E2 107.8052} C_DIS
LIN {X 91.2926,Y -31.3904,Z 100,A -23.9464,B 24.9307,C -1.9228,E1 25.1508,E2 109.26} C_DIS
LIN {X 90.3649,Y -33.9649,Z 100,A -25.4003,B 24.9306,C -1.9244,E1 25.1494,E2 110.702} C_DIS
LIN {X 89.5856,Y -35.9721,Z 100,A -26.7023,B 24.9309,C -1.9195,E1 25.1481,E2 112.0083} C_DIS
LIN {X 88.6782,Y -38.1544,Z 100,A -28.0955,B 24.9312,C -1.9156,E1 25.1465,E2 113.4031} C_DIS
LIN {X 87.7684,Y -40.2048,Z 100,A -29.4832,B 24.9317,C -1.9094,E1 25.1449,E2 114.798} C_DIS
LIN {X 86.6918,Y -42.4746,Z 100,A -31.0013,B 24.932,C -1.9039,E1 25.1431,E2 116.321} C_DIS
LIN {X 85.5979,Y -44.6377,Z 100,A -32.387,B 24.9322,C -1.9017,E1 25.1413,E2 117.7045} C_DIS
LIN {X 84.5515,Y -46.5908,Z 100,A -33.6951,B 24.9325,C -1.898,E1 25.1396,E2 119.0143} C_DIS
LIN {X 83.3953,Y -48.6304,Z 100,A -35.079,B 24.9327,C -1.8943,E1 25.1377,E2 120.3999} C_DIS
LIN {X 81.8987,Y -51.1074,Z 100,A -36.9108,B 24.9334,C -1.885,E1 25.135,E2 122.2442} C_DIS
LIN {X 80.2862,Y -53.6079,Z 100,A -38.7112,B 24.9338,C -1.8787,E1 25.1322,E2 124.0506} C_DIS
LIN {X 78.9268,Y -55.5902,Z 100,A -39.9638,B 24.9336,C -1.8814,E1 25.1302,E2 125.2907} C_DIS
LIN {X 77.4686,Y -57.6038,Z 100,A -41.5962,B 24.9344,C -1.8714,E1 25.1275,E2 126.9389} C_DIS
Enddeposition()
END
